KUKA KRL program: MyProgram_198().src

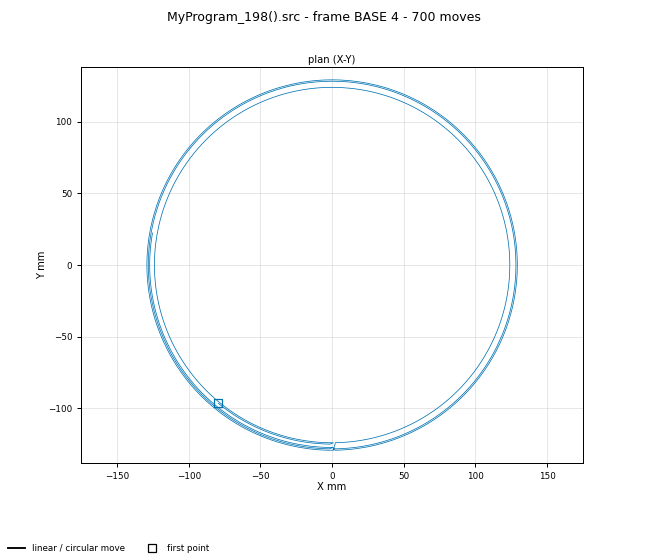
[picture p0: tool path of MyProgram_198().src in frame BASE 4, 700 of 700 moves have a stored position in this frame; points joined in program order, loops and branches not executed]
&ACCESS RVP
&REL 1
&PARAM TEMPLATE = C:\KRC\Roboter\Template\vorgabe
&PARAM EDITMASK = *
DEF MyProgram_198()
; ---- Setting reference (Base) ----
$BASE = BASE_DATA[4]

; --------------------------
; ---- Setting tool (TCP) ----
$TOOL = TOOL_DATA[3]
; --------------------------

$VEL.CP = VEL_APROX_PRINT
Startdeposition()
$VEL.CP = VEL_PRINT
LIN {X -79.3074,Y -96.5082,Z 142,A -131.7582,B 23.1277,C -1.1215,E1 23.053,E2 218.5929} C_DIS
LIN {X -76.0002,Y -99.1332,Z 142,A -129.8981,B 23.128,C -1.1147,E1 23.0571,E2 216.7428} C_DIS
LIN {X -73.2038,Y -101.2156,Z 142,A -128.0696,B 23.1276,C -1.1218,E1 23.0613,E2 214.889} C_DIS
LIN {X -68.9891,Y -104.1346,Z 142,A -125.8787,B 23.1281,C -1.111,E1 23.0663,E2 212.7178} C_DIS
LIN {X -65.7626,Y -106.2014,Z 142,A -124.3776,B 23.1288,C -1.0972,E1 23.0698,E2 211.2468} C_DIS
LIN {X -62.6284,Y -108.079,Z 142,A -122.461,B 23.1284,C -1.1052,E1 23.0744,E2 209.3034} C_DIS
LIN {X -59.0699,Y -110.0643,Z 142,A -120.3581,B 23.128,C -1.1129,E1 23.0796,E2 207.1744} C_DIS
LIN {X -55.3102,Y -111.9987,Z 142,A -118.661,B 23.1286,C -1.0998,E1 23.0838,E2 205.5056} C_DIS
LIN {X -52.0364,Y -113.5576,Z 142,A -116.9215,B 23.1286,C -1.1012,E1 23.0882,E2 203.7578} C_DIS
LIN {X -48.3423,Y -115.1781,Z 142,A -114.9515,B 23.1284,C -1.1045,E1 23.0933,E2 201.7745} C_DIS
LIN {X -44.2604,Y -116.8083,Z 142,A -113.1572,B 23.129,C -1.0928,E1 23.0979,E2 200.0059} C_DIS
LIN {X -41.267,Y -117.8988,Z 142,A -111.7171,B 23.129,C -1.0906,E1 23.1017,E2 198.5684} C_DIS
LIN {X -37.9757,Y -118.9992,Z 142,A -110.3261,B 23.1295,C -1.0804,E1 23.1053,E2 197.2004} C_DIS
LIN {X -34.3508,Y -120.098,Z 142,A -108.2397,B 23.1289,C -1.0946,E1 23.111,E2 195.0741} C_DIS
LIN {X -30.596,Y -121.1069,Z 142,A -106.5516,B 23.1291,C -1.0893,E1 23.1156,E2 193.3967} C_DIS
LIN {X -26.6613,Y -122.0338,Z 142,A -104.6727,B 23.1291,C -1.0895,E1 23.1207,E2 191.5148} C_DIS
LIN {X -23.1637,Y -122.7458,Z 142,A -102.9898,B 23.1291,C -1.0908,E1 23.1253,E2 189.8264} C_DIS
LIN {X -19.2282,Y -123.4232,Z 142,A -101.2648,B 23.1293,C -1.0855,E1 23.13,E2 188.1133} C_DIS
LIN {X -15.8715,Y -123.9001,Z 142,A -99.6847,B 23.1293,C -1.0863,E1 23.1344,E2 186.5299} C_DIS
LIN {X -11.9335,Y -124.3407,Z 142,A -97.8891,B 23.1293,C -1.0851,E1 23.1394,E2 184.7362} C_DIS
LIN {X -8.4853,Y -124.6251,Z 142,A -96.2436,B 23.1292,C -1.0876,E1 23.144,E2 183.0835} C_DIS
LIN {X -5.5832,Y -124.7887,Z 142,A -94.7991,B 23.129,C -1.0928,E1 23.1481,E2 181.6255} C_DIS
LIN {X -1.4686,Y -124.905,Z 142,A -92.9546,B 23.129,C -1.0911,E1 23.1532,E2 179.7852} C_DIS
LIN {X -1.4686,Y -124.905,Z 142,A -92.9546,B 23.129,C -1.0911,E1 23.1532,E2 179.7852} C_DIS
Enddeposition()
LIN {X 0.8717,Y -123.9392,Z 142,A -91.8325,B 22.3171,C -0.9594,E1 22.339,E2 178.8986} C_DIS
Startdeposition()
$VEL.CP = VEL_PRINT
LIN {X -2.2963,Y -123.9219,Z 142,A -93.916,B 22.3182,C -0.9325,E1 22.333,E2 181.0529} C_DIS
LIN {X -6.0852,Y -123.7935,Z 142,A -95.6272,B 22.3182,C -0.9341,E1 22.3282,E2 182.7603} C_DIS
LIN {X -9.1248,Y -123.6066,Z 142,A -97.0662,B 22.3182,C -0.9328,E1 22.3242,E2 184.2033} C_DIS
LIN {X -12.9239,Y -123.2677,Z 142,A -98.8033,B 22.3182,C -0.9341,E1 22.3194,E2 185.938} C_DIS
LIN {X -15.91,Y -122.9176,Z 142,A -100.1901,B 22.3182,C -0.9345,E1 22.3155,E2 187.3249} C_DIS
LIN {X -18.9628,Y -122.4836,Z 142,A -101.6065,B 22.3182,C -0.9352,E1 22.3116,E2 188.7406} C_DIS
LIN {X -21.9284,Y -121.9875,Z 142,A -103.0074,B 22.3182,C -0.9352,E1 22.3078,E2 190.1431} C_DIS
LIN {X -24.9422,Y -121.4073,Z 142,A -104.4213,B 22.3181,C -0.936,E1 22.3039,E2 191.5567} C_DIS
LIN {X -28.6367,Y -120.5898,Z 142,A -106.179,B 22.3181,C -0.9365,E1 22.2991,E2 193.3156} C_DIS
LIN {X -32.301,Y -119.6602,Z 142,A -107.9305,B 22.3181,C -0.9374,E1 22.2944,E2 195.0677} C_DIS
LIN {X -35.9945,Y -118.6012,Z 142,A -109.8524,B 22.3182,C -0.9326,E1 22.2892,E2 197.0059} C_DIS
LIN {X -40.3265,Y -117.199,Z 142,A -111.962,B 22.3182,C -0.9341,E1 22.2836,E2 199.116} C_DIS
LIN {X -43.9105,Y -115.9044,Z 142,A -113.5812,B 22.3178,C -0.9416,E1 22.2794,E2 200.7191} C_DIS
LIN {X -47.4374,Y -114.5057,Z 142,A -115.4966,B 22.318,C -0.9367,E1 22.2744,E2 202.6523} C_DIS
LIN {X -51.6487,Y -112.669,Z 142,A -117.6238,B 22.318,C -0.939,E1 22.269,E2 204.7794} C_DIS
LIN {X -55.3801,Y -110.8834,Z 142,A -119.4704,B 22.3178,C -0.944,E1 22.2644,E2 206.6182} C_DIS
LIN {X -58.4344,Y -109.3054,Z 142,A -120.9738,B 22.3175,C -0.9496,E1 22.2607,E2 208.1116} C_DIS
LIN {X -61.762,Y -107.4607,Z 142,A -122.9039,B 22.3177,C -0.945,E1 22.2559,E2 210.0601} C_DIS
LIN {X -65.6838,Y -105.1089,Z 142,A -125.0239,B 22.3176,C -0.9479,E1 22.2509,E2 212.1798} C_DIS
LIN {X -69.2138,Y -102.819,Z 142,A -126.9012,B 22.3174,C -0.9538,E1 22.2465,E2 214.0488} C_DIS
LIN {X -72.6168,Y -100.4441,Z 142,A -128.7387,B 22.3171,C -0.9603,E1 22.2424,E2 215.8762} C_DIS
LIN {X -75.6547,Y -98.1768,Z 142,A -130.6621,B 22.3172,C -0.9564,E1 22.238,E2 217.8175} C_DIS
LIN {X -79.2058,Y -95.3345,Z 142,A -132.6852,B 22.317,C -0.9636,E1 22.2337,E2 219.8305} C_DIS
LIN {X -82.3887,Y -92.5983,Z 142,A -134.734,B 22.317,C -0.963,E1 22.2293,E2 221.89} C_DIS
LIN {X -85.4698,Y -89.7616,Z 142,A -136.6617,B 22.3168,C -0.9673,E1 22.2254,E2 223.8153} C_DIS
LIN {X -88.7114,Y -86.5597,Z 142,A -138.7161,B 22.3165,C -0.9738,E1 22.2214,E2 225.8623} C_DIS
LIN {X -91.5742,Y -83.5252,Z 142,A -140.7246,B 22.3165,C -0.9749,E1 22.2176,E2 227.878} C_DIS
LIN {X -94.5817,Y -80.1033,Z 142,A -142.8001,B 22.3162,C -0.9809,E1 22.2138,E2 229.9482} C_DIS
LIN {X -96.7777,Y -77.4362,Z 142,A -144.4451,B 22.3162,C -0.9828,E1 22.2109,E2 231.597} C_DIS
LIN {X -99.5555,Y -73.8306,Z 142,A -146.5705,B 22.316,C -0.987,E1 22.2073,E2 233.7226} C_DIS
LIN {X -102.1996,Y -70.1244,Z 142,A -148.6828,B 22.3158,C -0.992,E1 22.2039,E2 235.8336} C_DIS
LIN {X -104.7148,Y -66.3102,Z 142,A -150.7774,B 22.3155,C -0.9981,E1 22.2007,E2 237.9239} C_DIS
LIN {X -106.7088,Y -63.0518,Z 142,A -152.5785,B 22.3154,C -1.0014,E1 22.1982,E2 239.7269} C_DIS
LIN {X -108.944,Y -59.1056,Z 142,A -154.6079,B 22.315,C -1.0097,E1 22.1954,E2 241.7464} C_DIS
LIN {X -110.5212,Y -56.0964,Z 142,A -156.1781,B 22.3148,C -1.0141,E1 22.1934,E2 243.3145} C_DIS
LIN {X -112.0468,Y -52.9856,Z 142,A -157.7322,B 22.3146,C -1.0204,E1 22.1915,E2 244.8615} C_DIS
LIN {X -113.6099,Y -49.5447,Z 142,A -159.6499,B 22.3146,C -1.0187,E1 22.1893,E2 246.7957} C_DIS
LIN {X -115.0085,Y -46.2039,Z 142,A -161.205,B 22.3142,C -1.0282,E1 22.1877,E2 248.3355} C_DIS
LIN {X -116.4356,Y -42.4819,Z 142,A -163.2031,B 22.3142,C -1.0275,E1 22.1857,E2 250.3482} C_DIS
LIN {X -117.9183,Y -38.1742,Z 142,A -165.3281,B 22.314,C -1.033,E1 22.1839,E2 252.4724} C_DIS
LIN {X -119.2482,Y -33.7908,Z 142,A -167.4478,B 22.3137,C -1.0393,E1 22.1822,E2 254.5893} C_DIS
LIN {X -120.2291,Y -30.1146,Z 142,A -169.1992,B 22.3135,C -1.045,E1 22.181,E2 256.3373} C_DIS
LIN {X -121.0983,Y -26.402,Z 142,A -170.8293,B 22.313,C -1.0555,E1 22.18,E2 257.9502} C_DIS
LIN {X -121.7047,Y -23.4477,Z 142,A -172.2411,B 22.3128,C -1.0592,E1 22.1792,E2 259.3619} C_DIS
LIN {X -122.2442,Y -20.449,Z 142,A -173.6444,B 22.3126,C -1.0637,E1 22.1785,E2 260.7624} C_DIS
LIN {X -122.7383,Y -17.2398,Z 142,A -175.2701,B 22.3126,C -1.0637,E1 22.1779,E2 262.3995} C_DIS
LIN {X -123.1888,Y -13.6572,Z 142,A -176.8563,B 22.3123,C -1.0721,E1 22.1774,E2 263.974} C_DIS
LIN {X -123.4861,Y -10.6336,Z 142,A -178.2667,B 22.3121,C -1.0763,E1 22.177,E2 265.3829} C_DIS
LIN {X -123.7095,Y -7.6032,Z 142,A -179.6751,B 22.3119,C -1.0806,E1 22.1767,E2 266.7895} C_DIS
LIN {X -123.8593,Y -4.5609,Z 142,A 178.7447,B 22.3119,C -1.0784,E1 22.1765,E2 268.3862} C_DIS
LIN {X -123.946,Y 0,Z 142,A 176.5529,B 22.3119,C -1.0819,E1 22.1765,E2 270.5837} C_DIS
LIN {X -123.8594,Y 4.5582,Z 142,A 174.6462,B 22.3111,C -1.0965,E1 22.1766,E2 272.4649} C_DIS
LIN {X -123.7172,Y 7.4784,Z 142,A 173.2388,B 22.3111,C -1.0986,E1 22.1768,E2 273.8762} C_DIS
LIN {X -123.4269,Y 11.3098,Z 142,A 171.3972,B 22.3109,C -1.1018,E1 22.1773,E2 275.7221} C_DIS
LIN {X -122.9987,Y 15.2809,Z 142,A 169.6572,B 22.3104,C -1.1118,E1 22.1778,E2 277.4473} C_DIS
LIN {X -122.5967,Y 18.2306,Z 142,A 168.2579,B 22.3102,C -1.1153,E1 22.1784,E2 278.8469} C_DIS
LIN {X -122.1586,Y 20.9622,Z 142,A 166.914,B 22.3102,C -1.1168,E1 22.179,E2 280.1957} C_DIS
LIN {X -121.5592,Y 24.1957,Z 142,A 165.4285,B 22.3099,C -1.123,E1 22.1798,E2 281.6749} C_DIS
LIN {X -120.93,Y 27.1649,Z 142,A 163.8565,B 22.3099,C -1.1209,E1 22.1807,E2 283.2629} C_DIS
LIN {X -119.8499,Y 31.5898,Z 142,A 161.7428,B 22.3097,C -1.1272,E1 22.1822,E2 285.3739} C_DIS
LIN {X -118.6079,Y 35.9727,Z 142,A 159.7772,B 22.3091,C -1.1392,E1 22.1837,E2 287.3206} C_DIS
LIN {X -117.6909,Y 38.8678,Z 142,A 158.2151,B 22.3091,C -1.1375,E1 22.185,E2 288.8976} C_DIS
LIN {X -116.4339,Y 42.4869,Z 142,A 156.5771,B 22.3087,C -1.148,E1 22.1866,E2 290.5181} C_DIS
LIN {X -115.0821,Y 46.0214,Z 142,A 154.664,B 22.3087,C -1.147,E1 22.1885,E2 292.446} C_DIS
LIN {X -113.3041,Y 50.2401,Z 142,A 152.519,B 22.3085,C -1.1523,E1 22.1909,E2 294.5905} C_DIS
LIN {X -111.72,Y 53.6698,Z 142,A 150.9241,B 22.3079,C -1.1633,E1 22.1928,E2 296.166} C_DIS
LIN {X -110.2395,Y 56.6497,Z 142,A 149.3135,B 22.3079,C -1.165,E1 22.1948,E2 297.7819} C_DIS
LIN {X -108.5935,Y 59.7474,Z 142,A 147.5881,B 22.3079,C -1.1657,E1 22.1971,E2 299.516} C_DIS
LIN {X -106.3109,Y 63.7204,Z 142,A 145.5115,B 22.3074,C -1.1733,E1 22.2,E2 301.5845} C_DIS
LIN {X -104.2933,Y 66.9711,Z 142,A 143.6733,B 22.3074,C -1.1755,E1 22.2028,E2 303.4275} C_DIS
LIN {X -101.7782,Y 70.7347,Z 142,A 141.5651,B 22.3071,C -1.1807,E1 22.2061,E2 305.5339} C_DIS
LIN {X -99.0918,Y 74.4518,Z 142,A 139.6016,B 22.3065,C -1.1925,E1 22.2093,E2 307.477} C_DIS
LIN {X -96.7618,Y 77.4562,Z 142,A 137.6837,B 22.3065,C -1.1908,E1 22.2126,E2 309.4096} C_DIS
LIN {X -94.1026,Y 80.6658,Z 142,A 135.7295,B 22.3063,C -1.1946,E1 22.2162,E2 311.3637} C_DIS
LIN {X -91.0649,Y 84.08,Z 142,A 133.6742,B 22.306,C -1.2021,E1 22.22,E2 313.4095} C_DIS
LIN {X -88.1717,Y 87.1095,Z 142,A 131.6512,B 22.306,C -1.2034,E1 22.2239,E2 315.4391} C_DIS
LIN {X -85.1819,Y 90.0348,Z 142,A 129.7181,B 22.3057,C -1.208,E1 22.2278,E2 317.3691} C_DIS
LIN {X -81.817,Y 93.1037,Z 142,A 127.6556,B 22.3053,C -1.2144,E1 22.2321,E2 319.424} C_DIS
LIN {X -78.9119,Y 95.5779,Z 142,A 125.9078,B 22.3051,C -1.2189,E1 22.2358,E2 321.1675} C_DIS
LIN {X -75.653,Y 98.1781,Z 142,A 123.875,B 22.3051,C -1.2188,E1 22.2403,E2 323.2091} C_DIS
LIN {X -71.9821,Y 100.8999,Z 142,A 121.7591,B 22.3049,C -1.2229,E1 22.2451,E2 325.3224} C_DIS
LIN {X -68.2096,Y 103.4874,Z 142,A 119.7612,B 22.3044,C -1.2317,E1 22.2497,E2 327.3049} C_DIS
LIN {X -64.9188,Y 105.583,Z 142,A 117.827,B 22.3045,C -1.2298,E1 22.2543,E2 329.2509} C_DIS
LIN {X -61.0554,Y 107.8637,Z 142,A 115.7414,B 22.3044,C -1.2329,E1 22.2593,E2 331.3353} C_DIS
LIN {X -57.2646,Y 109.9211,Z 142,A 113.8732,B 22.3039,C -1.2413,E1 22.2639,E2 333.1873} C_DIS
LIN {X -54.3534,Y 111.3899,Z 142,A 112.3781,B 22.3038,C -1.2441,E1 22.2676,E2 334.6793} C_DIS
LIN {X -51.6084,Y 112.6876,Z 142,A 110.971,B 22.3037,C -1.2461,E1 22.2712,E2 336.0852} C_DIS
LIN {X -48.1162,Y 114.2222,Z 142,A 109.0475,B 22.3039,C -1.2422,E1 22.2761,E2 338.0243} C_DIS
LIN {X -44.599,Y 115.6408,Z 142,A 107.3018,B 22.3037,C -1.2448,E1 22.2807,E2 339.7673} C_DIS
LIN {X -40.9841,Y 116.971,Z 142,A 105.5035,B 22.3037,C -1.2463,E1 22.2854,E2 341.5657} C_DIS
LIN {X -36.678,Y 118.392,Z 142,A 103.3984,B 22.3036,C -1.2483,E1 22.291,E2 343.6697} C_DIS
LIN {X -33.0611,Y 119.4523,Z 142,A 101.6561,B 22.3035,C -1.2501,E1 22.2957,E2 345.4105} C_DIS
LIN {X -28.6324,Y 120.5908,Z 142,A 99.5287,B 22.3034,C -1.2515,E1 22.3014,E2 347.5374} C_DIS
LIN {X -24.94,Y 121.4078,Z 142,A 97.9393,B 22.303,C -1.2595,E1 22.3057,E2 349.108} C_DIS
LIN {X -21.8511,Y 122.0014,Z 142,A 96.4534,B 22.303,C -1.2593,E1 22.3098,E2 350.5964} C_DIS
LIN {X -18.1786,Y 122.6042,Z 142,A 94.7493,B 22.3029,C -1.2611,E1 22.3145,E2 352.2975} C_DIS
LIN {X -15.1689,Y 123.0121,Z 142,A 93.1894,B 22.3032,C -1.2555,E1 22.3189,E2 353.8733} C_DIS
LIN {X -11.0173,Y 123.4536,Z 142,A 91.3043,B 22.303,C -1.2582,E1 22.3241,E2 355.7524} C_DIS
LIN {X -7.5913,Y 123.7102,Z 142,A 89.8371,B 22.3027,C -1.2639,E1 22.3281,E2 357.2053} C_DIS
LIN {X -4.5569,Y 123.8595,Z 142,A 88.2717,B 22.3031,C -1.2576,E1 22.3325,E2 358.7875} C_DIS
LIN {X -0.7453,Y 123.9408,Z 142,A 86.6712,B 22.3027,C -1.2647,E1 22.337,E2 360.3694} C_DIS
LIN {X 2.3024,Y 123.9218,Z 142,A 85.1012,B 22.303,C -1.2582,E1 22.3414,E2 361.9564} C_DIS
LIN {X 6.8655,Y 123.7543,Z 142,A 83.1554,B 22.3027,C -1.2651,E1 22.3468,E2 363.8832} C_DIS
LIN {X 9.895,Y 123.5484,Z 142,A 81.7369,B 22.3027,C -1.2644,E1 22.3507,E2 365.3028} C_DIS
LIN {X 12.9191,Y 123.2682,Z 142,A 80.2409,B 22.3029,C -1.2603,E1 22.3549,E2 366.8084} C_DIS
LIN {X 16.5992,Y 122.8272,Z 142,A 78.473,B 22.3031,C -1.2576,E1 22.3598,E2 368.5818} C_DIS
LIN {X 20.4296,Y 122.2475,Z 142,A 76.8358,B 22.3027,C -1.2635,E1 22.3643,E2 370.2016} C_DIS
LIN {X 23.5219,Y 121.6905,Z 142,A 75.2611,B 22.3031,C -1.2578,E1 22.3686,E2 371.7896} C_DIS
LIN {X 27.4214,Y 120.8714,Z 142,A 73.4485,B 22.3031,C -1.2581,E1 22.3736,E2 373.5987} C_DIS
LIN {X 31.608,Y 119.845,Z 142,A 71.4007,B 22.3032,C -1.2545,E1 22.3791,E2 375.6523} C_DIS
LIN {X 35.9885,Y 118.603,Z 142,A 69.3051,B 22.3032,C -1.2533,E1 22.3848,E2 377.7469} C_DIS
LIN {X 40.3212,Y 117.2009,Z 142,A 67.3524,B 22.303,C -1.2581,E1 22.3899,E2 379.6829} C_DIS
LIN {X 43.3345,Y 116.1202,Z 142,A 65.7635,B 22.3034,C -1.252,E1 22.3941,E2 381.2839} C_DIS
LIN {X 46.7481,Y 114.7892,Z 142,A 64.0309,B 22.3035,C -1.2486,E1 22.3986,E2 383.021} C_DIS
LIN {X 50.936,Y 112.9928,Z 142,A 62.0812,B 22.3033,C -1.253,E1 22.4035,E2 384.9539} C_DIS
LIN {X 53.6652,Y 111.7222,Z 142,A 60.6564,B 22.3035,C -1.2499,E1 22.4071,E2 386.3827} C_DIS
LIN {X 57.0846,Y 110.0156,Z 142,A 58.9614,B 22.3035,C -1.2507,E1 22.4113,E2 388.0703} C_DIS
LIN {X 60.4301,Y 108.2151,Z 142,A 57.0274,B 22.304,C -1.2405,E1 22.4161,E2 390.0246} C_DIS
LIN {X 64.3888,Y 105.9073,Z 142,A 54.9005,B 22.3042,C -1.237,E1 22.4212,E2 392.1533} C_DIS
LIN {X 68.2553,Y 103.4573,Z 142,A 52.8091,B 22.3042,C -1.2347,E1 22.4261,E2 394.243} C_DIS
LIN {X 71.9872,Y 100.8962,Z 142,A 50.7274,B 22.3044,C -1.2316,E1 22.4309,E2 396.3246} C_DIS
LIN {X 75.6425,Y 98.1863,Z 142,A 48.6243,B 22.3046,C -1.2279,E1 22.4356,E2 398.4288} C_DIS
LIN {X 79.2139,Y 95.3278,Z 142,A 46.6078,B 22.3046,C -1.2282,E1 22.4399,E2 400.4358} C_DIS
LIN {X 82.4003,Y 92.588,Z 142,A 44.5842,B 22.305,C -1.2208,E1 22.4442,E2 402.4698} C_DIS
LIN {X 85.4671,Y 89.7642,Z 142,A 42.6802,B 22.3052,C -1.2179,E1 22.4481,E2 404.3726} C_DIS
LIN {X 88.7091,Y 86.5621,Z 142,A 40.6465,B 22.3052,C -1.2166,E1 22.4521,E2 406.3999} C_DIS
LIN {X 91.5695,Y 83.5304,Z 142,A 38.6578,B 22.3056,C -1.2095,E1 22.4559,E2 408.3972} C_DIS
LIN {X 94.591,Y 80.0924,Z 142,A 36.6269,B 22.3056,C -1.2084,E1 22.4596,E2 410.4206} C_DIS
LIN {X 97.2514,Y 76.8407,Z 142,A 34.6896,B 22.3059,C -1.204,E1 22.463,E2 412.3592} C_DIS
LIN {X 99.5507,Y 73.837,Z 142,A 32.8768,B 22.3062,C -1.1969,E1 22.466,E2 414.1809} C_DIS
LIN {X 102.2052,Y 70.1163,Z 142,A 30.783,B 22.3065,C -1.1924,E1 22.4694,E2 416.2748} C_DIS
LIN {X 104.4189,Y 66.775,Z 142,A 28.9924,B 22.3065,C -1.1904,E1 22.4721,E2 418.0605} C_DIS
LIN {X 106.719,Y 63.0344,Z 142,A 26.9374,B 22.3069,C -1.1839,E1 22.4751,E2 420.1206} C_DIS
LIN {X 108.9413,Y 59.1106,Z 142,A 24.9414,B 22.3069,C -1.1823,E1 22.4778,E2 422.1091} C_DIS
LIN {X 110.3519,Y 56.4289,Z 142,A 23.6107,B 22.307,C -1.1816,E1 22.4795,E2 423.4336} C_DIS
LIN {X 111.7602,Y 53.5856,Z 142,A 22.0436,B 22.3074,C -1.173,E1 22.4814,E2 425.0138} C_DIS
LIN {X 113.3091,Y 50.2289,Z 142,A 20.4626,B 22.3074,C -1.1739,E1 22.4832,E2 426.5826} C_DIS
LIN {X 114.7964,Y 46.73,Z 142,A 18.555,B 22.308,C -1.162,E1 22.4853,E2 428.5093} C_DIS
LIN {X 116.4347,Y 42.4845,Z 142,A 16.4589,B 22.3083,C -1.1562,E1 22.4873,E2 430.6074} C_DIS
LIN {X 117.9158,Y 38.1821,Z 142,A 14.5324,B 22.3082,C -1.1579,E1 22.489,E2 432.517} C_DIS
LIN {X 118.9989,Y 34.6564,Z 142,A 12.8155,B 22.3085,C -1.1523,E1 22.4904,E2 434.2377} C_DIS
LIN {X 120.0323,Y 30.8902,Z 142,A 10.8916,B 22.309,C -1.1414,E1 22.4918,E2 436.1774} C_DIS
LIN {X 121.0928,Y 26.4273,Z 142,A 8.9201,B 22.309,C -1.1416,E1 22.493,E2 438.1353} C_DIS
LIN {X 121.8497,Y 22.6894,Z 142,A 7.0741,B 22.3094,C -1.1324,E1 22.494,E2 439.9934} C_DIS
LIN {X 122.4848,Y 18.955,Z 142,A 5.425,B 22.3094,C -1.1315,E1 22.4948,E2 441.6337} C_DIS
LIN {X 123.0119,Y 15.1704,Z 142,A 3.6994,B 22.3097,C -1.1278,E1 22.4954,E2 443.3574} C_DIS
LIN {X 123.3462,Y 12.1505,Z 142,A 2.3087,B 22.3098,C -1.124,E1 22.4958,E2 444.7488} C_DIS
LIN {X 123.621,Y 8.9269,Z 142,A 0.7565,B 22.3102,C -1.1167,E1 22.4961,E2 446.3096} C_DIS
LIN {X 123.8594,Y 4.5572,Z 142,A -1.3319,B 22.3106,C -1.1073,E1 22.4964,E2 448.4087} C_DIS
LIN {X 123.9459,Y 0.017,Z 142,A -3.3195,B 22.3107,C -1.1056,E1 22.4964,E2 450.3872} C_DIS
LIN {X 123.9065,Y -3.0353,Z 142,A -4.6782,B 22.3108,C -1.1035,E1 22.4964,E2 451.7422} C_DIS
LIN {X 123.7935,Y -6.0869,Z 142,A -6.0652,B 22.311,C -1.1001,E1 22.4962,E2 453.1288} C_DIS
LIN {X 123.5826,Y -9.4536,Z 142,A -7.6911,B 22.3113,C -1.092,E1 22.4959,E2 454.7649} C_DIS
LIN {X 123.2685,Y -12.9166,Z 142,A -9.2129,B 22.3113,C -1.0908,E1 22.4955,E2 456.2796} C_DIS
LIN {X 122.8178,Y -16.671,Z 142,A -10.9283,B 22.3116,C -1.0867,E1 22.4949,E2 457.9943} C_DIS
LIN {X 122.3704,Y -19.6926,Z 142,A -12.3232,B 22.3118,C -1.083,E1 22.4943,E2 459.3897} C_DIS
LIN {X 121.812,Y -22.8863,Z 142,A -13.9781,B 22.3123,C -1.0711,E1 22.4935,E2 461.0647} C_DIS
LIN {X 120.9197,Y -27.21,Z 142,A -16.008,B 22.3126,C -1.0651,E1 22.4923,E2 463.0968} C_DIS
LIN {X 119.8492,Y -31.5924,Z 142,A -18.0816,B 22.3128,C -1.0591,E1 22.4909,E2 465.1727} C_DIS
LIN {X 118.604,Y -35.9854,Z 142,A -20.0205,B 22.3128,C -1.0603,E1 22.4894,E2 467.0958} C_DIS
LIN {X 117.6877,Y -38.8773,Z 142,A -21.4155,B 22.313,C -1.0563,E1 22.4882,E2 468.4922} C_DIS
LIN {X 116.6962,Y -41.7592,Z 142,A -22.9368,B 22.3134,C -1.0468,E1 22.4867,E2 470.0288} C_DIS
LIN {X 115.3575,Y -45.3276,Z 142,A -24.7206,B 22.3137,C -1.0404,E1 22.4849,E2 471.8181} C_DIS
LIN {X 113.6147,Y -49.5335,Z 142,A -26.7981,B 22.3139,C -1.0353,E1 22.4827,E2 473.8961} C_DIS
LIN {X 111.9515,Y -53.1852,Z 142,A -28.6043,B 22.3141,C -1.032,E1 22.4805,E2 475.6999} C_DIS
LIN {X 110.3004,Y -56.5301,Z 142,A -30.2933,B 22.3142,C -1.0285,E1 22.4784,E2 477.3878} C_DIS
LIN {X 108.581,Y -59.77,Z 142,A -32.0443,B 22.3145,C -1.021,E1 22.4761,E2 479.1479} C_DIS
LIN {X 106.3109,Y -63.7204,Z 142,A -34.1443,B 22.3148,C -1.0152,E1 22.4731,E2 481.2507} C_DIS
LIN {X 103.8834,Y -67.6051,Z 142,A -36.2396,B 22.315,C -1.0103,E1 22.47,E2 483.347} C_DIS
LIN {X 101.3314,Y -71.3733,Z 142,A -38.3243,B 22.3152,C -1.0054,E1 22.4667,E2 485.4329} C_DIS
LIN {X 98.6425,Y -75.0463,Z 142,A -40.4278,B 22.3154,C -0.9998,E1 22.4631,E2 487.5397} C_DIS
LIN {X 95.7941,Y -78.6496,Z 142,A -42.4577,B 22.3155,C -0.9984,E1 22.4596,E2 489.5625} C_DIS
LIN {X 93.1031,Y -81.8177,Z 142,A -44.3785,B 22.3157,C -0.9935,E1 22.4561,E2 491.4862} C_DIS
LIN {X 90.5128,Y -84.6741,Z 142,A -46.1372,B 22.3159,C -0.9902,E1 22.4528,E2 493.245} C_DIS
LIN {X 87.6214,Y -87.6631,Z 142,A -48.129,B 22.3162,C -0.9824,E1 22.4488,E2 495.2475} C_DIS
LIN {X 84.6231,Y -90.5603,Z 142,A -50.0304,B 22.3163,C -0.979,E1 22.445,E2 497.1488} C_DIS
LIN {X 81.216,Y -93.6284,Z 142,A -52.157,B 22.3165,C -0.9738,E1 22.4405,E2 499.2794} C_DIS
LIN {X 78.0288,Y -96.3004,Z 142,A -54.0561,B 22.3167,C -0.9707,E1 22.4364,E2 501.1785} C_DIS
LIN {X 74.453,Y -99.0909,Z 142,A -56.1566,B 22.3169,C -0.9661,E1 22.4318,E2 503.2824} C_DIS
LIN {X 70.743,Y -101.7724,Z 142,A -58.2583,B 22.317,C -0.9624,E1 22.427,E2 505.3854} C_DIS
LIN {X 66.9581,Y -104.3016,Z 142,A -60.3509,B 22.3171,C -0.9589,E1 22.4221,E2 507.4794} C_DIS
LIN {X 63.0567,Y -106.7059,Z 142,A -62.4551,B 22.3173,C -0.9557,E1 22.4171,E2 509.5846} C_DIS
LIN {X 59.118,Y -108.9373,Z 142,A -64.5655,B 22.3175,C -0.9512,E1 22.4119,E2 511.6996} C_DIS
LIN {X 55.2848,Y -110.9304,Z 142,A -66.4642,B 22.3175,C -0.9523,E1 22.4072,E2 513.5895} C_DIS
LIN {X 51.6616,Y -112.663,Z 142,A -68.2372,B 22.3174,C -0.9532,E1 22.4027,E2 515.3552} C_DIS
LIN {X 48.1088,Y -114.2253,Z 142,A -70.1701,B 22.3177,C -0.9444,E1 22.3977,E2 517.3058} C_DIS
LIN {X 43.9118,Y -115.9039,Z 142,A -72.1075,B 22.3176,C -0.9483,E1 22.3927,E2 519.2283} C_DIS
LIN {X 40.3106,Y -117.2045,Z 142,A -74.0028,B 22.3179,C -0.9405,E1 22.3877,E2 521.1394} C_DIS
LIN {X 36.7007,Y -118.3851,Z 142,A -75.7769,B 22.318,C -0.9377,E1 22.383,E2 522.9173} C_DIS
LIN {X 33.0811,Y -119.4467,Z 142,A -77.354,B 22.3178,C -0.9431,E1 22.3788,E2 524.4773} C_DIS
LIN {X 29.3499,Y -120.4179,Z 142,A -79.1334,B 22.3178,C -0.9414,E1 22.374,E2 526.2579} C_DIS
LIN {X 25.665,Y -121.2574,Z 142,A -80.8674,B 22.3178,C -0.9404,E1 22.3692,E2 527.992} C_DIS
LIN {X 22.6853,Y -121.8505,Z 142,A -82.2664,B 22.3179,C -0.9395,E1 22.3654,E2 529.3915} C_DIS
LIN {X 19.214,Y -122.4447,Z 142,A -83.9711,B 22.3181,C -0.935,E1 22.3607,E2 531.1061} C_DIS
LIN {X 15.3695,Y -122.9881,Z 142,A -85.7751,B 22.3181,C -0.9335,E1 22.3557,E2 532.9124} C_DIS
LIN {X 12.1455,Y -123.3467,Z 142,A -87.1981,B 22.3181,C -0.936,E1 22.3518,E2 534.3277} C_DIS
LIN {X 8.8298,Y -123.6281,Z 142,A -88.793,B 22.3181,C -0.9328,E1 22.3473,E2 535.93} C_DIS
LIN {X 5.287,Y -123.831,Z 142,A -90.3796,B 22.3181,C -0.9345,E1 22.3429,E2 537.5115} C_DIS
LIN {X 2.2861,Y -123.9221,Z 142,A -91.7661,B 22.3181,C -0.9342,E1 22.339,E2 538.8986} C_DIS
LIN {X 2.2861,Y -123.9221,Z 142,A -91.7661,B 22.3181,C -0.9342,E1 22.339,E2 538.8986} C_DIS
Enddeposition()
LIN {X 0.9159,Y -129.1721,Z 143,A -92.6978,B 24.9656,C -1.3555,E1 25.0017,E2 539.1265} C_DIS
Startdeposition()
$VEL.CP = VEL_PRINT
LIN {X -2.056,Y -129.1619,Z 143,A -94.4314,B 24.9667,C -1.3341,E1 24.9968,E2 540.9106} C_DIS
LIN {X -5.4479,Y -129.064,Z 143,A -95.9238,B 24.9667,C -1.3346,E1 24.9926,E2 542.4023} C_DIS
LIN {X -9.2404,Y -128.8474,Z 143,A -97.6422,B 24.9667,C -1.3329,E1 24.9878,E2 544.1253} C_DIS
LIN {X -12.7283,Y -128.5501,Z 143,A -99.1732,B 24.9667,C -1.334,E1 24.9835,E2 545.6542} C_DIS
LIN {X -16.3368,Y -128.1417,Z 143,A -100.8519,B 24.9668,C -1.3309,E1 24.9789,E2 547.3415} C_DIS
LIN {X -19.8619,Y -127.642,Z 143,A -102.343,B 24.9666,C -1.3357,E1 24.9748,E2 548.8224} C_DIS
LIN {X -22.8537,Y -127.1404,Z 143,A -103.6917,B 24.9666,C -1.336,E1 24.9711,E2 550.1718} C_DIS
LIN {X -25.8549,Y -126.5642,Z 143,A -105.0506,B 24.9666,C -1.3364,E1 24.9673,E2 551.5314} C_DIS
LIN {X -28.9111,Y -125.9012,Z 143,A -106.4793,B 24.9666,C -1.335,E1 24.9634,E2 552.9651} C_DIS
LIN {X -32.1688,Y -125.109,Z 143,A -107.9331,B 24.9665,C -1.3375,E1 24.9595,E2 554.4151} C_DIS
LIN {X -35.1544,Y -124.303,Z 143,A -109.3333,B 24.9665,C -1.337,E1 24.9557,E2 555.8187} C_DIS
LIN {X -38.1245,Y -123.4243,Z 143,A -110.714,B 24.9665,C -1.3377,E1 24.952,E2 557.2001} C_DIS
LIN {X -41.0909,Y -122.4685,Z 143,A -112.1194,B 24.9665,C -1.3377,E1 24.9483,E2 558.6082} C_DIS
LIN {X -44.1762,Y -121.3899,Z 143,A -113.5097,B 24.9663,C -1.3418,E1 24.9447,E2 559.9913} C_DIS
LIN {X -47.0009,Y -120.324,Z 143,A -114.8983,B 24.9663,C -1.3407,E1 24.941,E2 561.3855} C_DIS
LIN {X -50.1973,Y -119.0266,Z 143,A -116.3763,B 24.9661,C -1.3449,E1 24.9372,E2 562.857} C_DIS
LIN {X -52.9783,Y -117.8145,Z 143,A -117.7771,B 24.9661,C -1.3437,E1 24.9336,E2 564.2639} C_DIS
LIN {X -55.9912,Y -116.413,Z 143,A -119.242,B 24.9661,C -1.3459,E1 24.9299,E2 565.7273} C_DIS
LIN {X -59.3318,Y -114.7488,Z 143,A -120.895,B 24.966,C -1.3481,E1 24.9258,E2 567.3795} C_DIS
LIN {X -62.0674,Y -113.2919,Z 143,A -122.3372,B 24.966,C -1.3467,E1 24.9223,E2 568.8291} C_DIS
LIN {X -65.7504,Y -111.1953,Z 143,A -124.2414,B 24.966,C -1.3482,E1 24.9177,E2 570.7353} C_DIS
LIN {X -69.2992,Y -109.0191,Z 143,A -126.1244,B 24.9659,C -1.3493,E1 24.9132,E2 572.6217} C_DIS
LIN {X -72.7546,Y -106.7441,Z 143,A -127.9389,B 24.9657,C -1.3533,E1 24.909,E2 574.4326} C_DIS
LIN {X -76.1455,Y -104.3523,Z 143,A -129.8434,B 24.9657,C -1.3534,E1 24.9047,E2 576.3436} C_DIS
LIN {X -79.5443,Y -101.7849,Z 143,A -131.7274,B 24.9655,C -1.3571,E1 24.9005,E2 578.2255} C_DIS
LIN {X -82.9887,Y -98.9962,Z 143,A -133.656,B 24.9652,C -1.3627,E1 24.8963,E2 580.1483} C_DIS
LIN {X -86.0043,Y -96.3882,Z 143,A -135.4758,B 24.9652,C -1.3638,E1 24.8925,E2 581.9727} C_DIS
LIN {X -89.2124,Y -93.4265,Z 143,A -137.3778,B 24.9649,C -1.3695,E1 24.8887,E2 583.8689} C_DIS
LIN {X -92.1442,Y -90.5364,Z 143,A -139.2175,B 24.9647,C -1.3728,E1 24.885,E2 585.7086} C_DIS
LIN {X -95.0674,Y -87.4617,Z 143,A -141.1028,B 24.9645,C -1.3768,E1 24.8814,E2 587.5924} C_DIS
LIN {X -97.7978,Y -84.3977,Z 143,A -142.9421,B 24.9643,C -1.3802,E1 24.878,E2 589.4321} C_DIS
LIN {X -100.3934,Y -81.2933,Z 143,A -144.781,B 24.9643,C -1.3824,E1 24.8748,E2 591.2742} C_DIS
LIN {X -103.1453,Y -77.7716,Z 143,A -146.7048,B 24.9638,C -1.3901,E1 24.8715,E2 593.189} C_DIS
LIN {X -105.593,Y -74.4143,Z 143,A -148.5941,B 24.9637,C -1.3926,E1 24.8684,E2 595.0815} C_DIS
LIN {X -108.1233,Y -70.6887,Z 143,A -150.6532,B 24.9636,C -1.3949,E1 24.8652,E2 597.1453} C_DIS
LIN {X -110.5126,Y -66.8905,Z 143,A -152.5862,B 24.9631,C -1.4029,E1 24.8624,E2 599.0691} C_DIS
LIN {X -112.6373,Y -63.2473,Z 143,A -154.4442,B 24.9628,C -1.4087,E1 24.8598,E2 600.9231} C_DIS
LIN {X -114.6313,Y -59.5554,Z 143,A -156.2326,B 24.9624,C -1.4173,E1 24.8575,E2 602.7004} C_DIS
LIN {X -115.9907,Y -56.8607,Z 143,A -157.6515,B 24.9624,C -1.4173,E1 24.8557,E2 604.1268} C_DIS
LIN {X -117.3701,Y -53.9558,Z 143,A -159.0627,B 24.9621,C -1.4222,E1 24.8541,E2 605.5342} C_DIS
LIN {X -118.7433,Y -50.8635,Z 143,A -160.5441,B 24.9618,C -1.4275,E1 24.8524,E2 607.0112} C_DIS
LIN {X -119.9639,Y -47.9137,Z 143,A -161.9681,B 24.9616,C -1.4313,E1 24.8509,E2 608.434} C_DIS
LIN {X -121.2134,Y -44.6621,Z 143,A -163.5143,B 24.9614,C -1.4359,E1 24.8494,E2 609.978} C_DIS
LIN {X -122.134,Y -42.0745,Z 143,A -164.8037,B 24.9614,C -1.4363,E1 24.8482,E2 611.2738} C_DIS
LIN {X -123.292,Y -38.5568,Z 143,A -166.4004,B 24.961,C -1.4434,E1 24.8468,E2 612.8627} C_DIS
LIN {X -124.1938,Y -35.545,Z 143,A -167.8019,B 24.9608,C -1.4474,E1 24.8457,E2 614.2628} C_DIS
LIN {X -125.2569,Y -31.5861,Z 143,A -169.6431,B 24.9605,C -1.452,E1 24.8444,E2 616.1037} C_DIS
LIN {X -125.956,Y -28.6712,Z 143,A -170.9863,B 24.9603,C -1.4556,E1 24.8436,E2 617.4462} C_DIS
LIN {X -126.7368,Y -25.0066,Z 143,A -172.6367,B 24.96,C -1.4614,E1 24.8427,E2 619.0926} C_DIS
LIN {X -127.1856,Y -22.6012,Z 143,A -173.7503,B 24.9599,C -1.4636,E1 24.8421,E2 620.2076} C_DIS
LIN {X -127.7607,Y -19.0953,Z 143,A -175.3051,B 24.9595,C -1.4696,E1 24.8414,E2 621.7572} C_DIS
LIN {X -128.2196,Y -15.7127,Z 143,A -176.9142,B 24.9595,C -1.4701,E1 24.8408,E2 623.3748} C_DIS
LIN {X -128.5897,Y -12.3156,Z 143,A -178.3686,B 24.9591,C -1.4779,E1 24.8404,E2 624.8194} C_DIS
LIN {X -128.8707,Y -8.9214,Z 143,A 179.9612,B 24.9592,C -1.4754,E1 24.8401,E2 626.5054} C_DIS
LIN {X -129.0837,Y -4.9409,Z 143,A 178.2793,B 24.9587,C -1.4852,E1 24.8399,E2 628.1742} C_DIS
LIN {X -129.1779,Y -0.7281,Z 143,A 176.5535,B 24.958,C -1.4979,E1 24.8398,E2 629.88} C_DIS
LIN {X -129.1484,Y 2.8673,Z 143,A 174.6921,B 24.9584,C -1.4909,E1 24.8398,E2 631.7694} C_DIS
LIN {X -129.0162,Y 6.4677,Z 143,A 173.2186,B 24.9577,C -1.5019,E1 24.84,E2 633.2255} C_DIS
LIN {X -128.8182,Y 9.6396,Z 143,A 171.6973,B 24.9577,C -1.5014,E1 24.8403,E2 634.7572} C_DIS
LIN {X -128.447,Y 13.7243,Z 143,A 169.9891,B 24.9571,C -1.5125,E1 24.8408,E2 636.4492} C_DIS
LIN {X -128.0706,Y 16.8793,Z 143,A 168.6059,B 24.9568,C -1.5183,E1 24.8413,E2 637.8267} C_DIS
LIN {X -127.642,Y 19.8619,Z 143,A 167.2193,B 24.9567,C -1.5204,E1 24.8418,E2 639.2165} C_DIS
LIN {X -127.1488,Y 22.8066,Z 143,A 165.8698,B 24.9565,C -1.5236,E1 24.8425,E2 640.5665} C_DIS
LIN {X -126.4956,Y 26.1918,Z 143,A 164.3438,B 24.9562,C -1.5287,E1 24.8433,E2 642.0893} C_DIS
LIN {X -125.7625,Y 29.5184,Z 143,A 162.8181,B 24.956,C -1.5329,E1 24.8443,E2 643.6139} C_DIS
LIN {X -125.124,Y 32.1099,Z 143,A 161.6132,B 24.9558,C -1.5358,E1 24.8451,E2 644.819} C_DIS
LIN {X -124.2571,Y 35.3187,Z 143,A 160.13,B 24.9556,C -1.5402,E1 24.8462,E2 646.3005} C_DIS
LIN {X -123.292,Y 38.5568,Z 143,A 158.6267,B 24.9553,C -1.5447,E1 24.8474,E2 647.8016} C_DIS
LIN {X -122.392,Y 41.3207,Z 143,A 157.3124,B 24.9551,C -1.5477,E1 24.8486,E2 649.1162} C_DIS
LIN {X -121.2507,Y 44.5625,Z 143,A 155.7902,B 24.9548,C -1.5526,E1 24.85,E2 650.6354} C_DIS
LIN {X -120.3028,Y 47.0554,Z 143,A 154.5682,B 24.9548,C -1.5546,E1 24.8512,E2 651.8597} C_DIS
LIN {X -119.1061,Y 50.0069,Z 143,A 153.1534,B 24.9545,C -1.5589,E1 24.8527,E2 653.2721} C_DIS
LIN {X -117.8285,Y 52.9469,Z 143,A 151.726,B 24.9542,C -1.563,E1 24.8543,E2 654.6975} C_DIS
LIN {X -116.2564,Y 56.3189,Z 143,A 150.0863,B 24.9539,C -1.5685,E1 24.8563,E2 656.333} C_DIS
LIN {X -114.8669,Y 59.0997,Z 143,A 148.6757,B 24.9537,C -1.5712,E1 24.8581,E2 657.7447} C_DIS
LIN {X -113.0365,Y 62.5309,Z 143,A 146.8533,B 24.9537,C -1.5718,E1 24.8605,E2 659.5752} C_DIS
LIN {X -110.7887,Y 66.4331,Z 143,A 144.8237,B 24.9534,C -1.5762,E1 24.8634,E2 661.6048} C_DIS
LIN {X -108.5736,Y 69.9951,Z 143,A 142.9857,B 24.9531,C -1.5826,E1 24.8661,E2 663.4369} C_DIS
LIN {X -106.275,Y 73.4381,Z 143,A 141.0995,B 24.9529,C -1.5855,E1 24.8691,E2 665.3256} C_DIS
LIN {X -103.7633,Y 76.9455,Z 143,A 139.1694,B 24.9526,C -1.5901,E1 24.8723,E2 667.2542} C_DIS
LIN {X -101.1059,Y 80.405,Z 143,A 137.2778,B 24.9522,C -1.5973,E1 24.8755,E2 669.1375} C_DIS
LIN {X -98.3881,Y 83.7087,Z 143,A 135.3825,B 24.9519,C -1.6025,E1 24.8789,E2 671.0293} C_DIS
LIN {X -95.7067,Y 86.7618,Z 143,A 133.5496,B 24.9517,C -1.6057,E1 24.8823,E2 672.8626} C_DIS
LIN {X -92.8819,Y 89.7794,Z 143,A 131.693,B 24.9515,C -1.6092,E1 24.8859,E2 674.7189} C_DIS
LIN {X -89.8928,Y 92.7721,Z 143,A 129.8186,B 24.9512,C -1.6139,E1 24.8896,E2 676.5901} C_DIS
LIN {X -86.8984,Y 95.5827,Z 143,A 127.9763,B 24.951,C -1.6173,E1 24.8934,E2 678.4319} C_DIS
LIN {X -83.7087,Y 98.3881,Z 143,A 126.0947,B 24.9507,C -1.6217,E1 24.8973,E2 680.3102} C_DIS
LIN {X -80.405,Y 101.1059,Z 143,A 124.2112,B 24.9504,C -1.6266,E1 24.9014,E2 682.1892} C_DIS
LIN {X -77.1058,Y 103.6439,Z 143,A 122.3574,B 24.9502,C -1.6302,E1 24.9055,E2 684.0412} C_DIS
LIN {X -73.8226,Y 106.0075,Z 143,A 120.5339,B 24.9501,C -1.6325,E1 24.9097,E2 685.8653} C_DIS
LIN {X -70.3867,Y 108.3193,Z 143,A 118.6905,B 24.9499,C -1.6359,E1 24.914,E2 687.7069} C_DIS
LIN {X -66.9381,Y 110.4838,Z 143,A 116.8666,B 24.9497,C -1.6384,E1 24.9183,E2 689.5304} C_DIS
LIN {X -63.3674,Y 112.5698,Z 143,A 115.0347,B 24.9495,C -1.6419,E1 24.9227,E2 691.3596} C_DIS
LIN {X -59.6528,Y 114.5802,Z 143,A 113.2515,B 24.949,C -1.6494,E1 24.9271,E2 693.1299} C_DIS
LIN {X -56.6984,Y 116.0708,Z 143,A 111.7512,B 24.949,C -1.6502,E1 24.9308,E2 694.6321} C_DIS
LIN {X -53.9468,Y 117.3743,Z 143,A 110.3629,B 24.949,C -1.6506,E1 24.9344,E2 696.0231} C_DIS
LIN {X -50.5246,Y 118.8899,Z 143,A 108.7482,B 24.9487,C -1.6552,E1 24.9385,E2 697.6307} C_DIS
LIN {X -47.5506,Y 120.1103,Z 143,A 107.3196,B 24.9485,C -1.6571,E1 24.9422,E2 699.0579} C_DIS
LIN {X -44.5625,Y 121.2507,Z 143,A 105.8986,B 24.9485,C -1.6588,E1 24.9459,E2 700.4777} C_DIS
LIN {X -40.8005,Y 122.5652,Z 143,A 104.1196,B 24.9483,C -1.6605,E1 24.9506,E2 702.256} C_DIS
LIN {X -37.7067,Y 123.5521,Z 143,A 102.6833,B 24.9483,C -1.6624,E1 24.9544,E2 703.6904} C_DIS
LIN {X -34.6942,Y 124.4317,Z 143,A 101.2765,B 24.9482,C -1.6632,E1 24.9582,E2 705.0975} C_DIS
LIN {X -31.3616,Y 125.3139,Z 143,A 99.7445,B 24.9481,C -1.6646,E1 24.9623,E2 706.6285} C_DIS
LIN {X -28.4576,Y 126.0048,Z 143,A 98.4452,B 24.9479,C -1.667,E1 24.9659,E2 707.9238} C_DIS
LIN {X -25.625,Y 126.6109,Z 143,A 97.1162,B 24.9479,C -1.666,E1 24.9695,E2 709.2567} C_DIS
LIN {X -22.6078,Y 127.1844,Z 143,A 95.7428,B 24.9479,C -1.6665,E1 24.9733,E2 710.6302} C_DIS
LIN {X -19.4781,Y 127.7014,Z 143,A 94.377,B 24.9478,C -1.6695,E1 24.977,E2 711.9902} C_DIS
LIN {X -15.709,Y 128.22,Z 143,A 92.6183,B 24.9479,C -1.6671,E1 24.9819,E2 713.756} C_DIS
LIN {X -12.2493,Y 128.5961,Z 143,A 91.1556,B 24.9476,C -1.6719,E1 24.9859,E2 715.2082} C_DIS
LIN {X -8.9248,Y 128.8704,Z 143,A 89.6624,B 24.9476,C -1.6719,E1 24.9901,E2 716.7021} C_DIS
LIN {X -5.7589,Y 129.0518,Z 143,A 88.0981,B 24.9481,C -1.6646,E1 24.9945,E2 718.284} C_DIS
LIN {X -2.056,Y 129.1619,Z 143,A 86.601,B 24.9476,C -1.6723,E1 24.9986,E2 719.7631} C_DIS
LIN {X 1.8756,Y 129.1649,Z 143,A 84.8047,B 24.9477,C -1.67,E1 25.0037,E2 721.5647} C_DIS
LIN {X 5.7589,Y 129.0518,Z 143,A 83.1296,B 24.9476,C -1.6725,E1 25.0083,E2 723.2334} C_DIS
LIN {X 9.3107,Y 128.8422,Z 143,A 81.577,B 24.9476,C -1.6737,E1 25.0127,E2 724.7824} C_DIS
LIN {X 12.2493,Y 128.5961,Z 143,A 80.2285,B 24.9476,C -1.6716,E1 25.0164,E2 726.1352} C_DIS
LIN {X 15.2057,Y 128.2801,Z 143,A 78.9077,B 24.9476,C -1.6713,E1 25.0201,E2 727.4559} C_DIS
LIN {X 18.1778,Y 127.8927,Z 143,A 77.5763,B 24.9476,C -1.6708,E1 25.0238,E2 728.7871} C_DIS
LIN {X 21.3565,Y 127.4005,Z 143,A 76.1869,B 24.9476,C -1.6722,E1 25.0276,E2 730.1719} C_DIS
LIN {X 24.3533,Y 126.8617,Z 143,A 74.8162,B 24.9476,C -1.6707,E1 25.0313,E2 731.5447} C_DIS
LIN {X 27.6421,Y 126.1864,Z 143,A 73.3199,B 24.9478,C -1.6696,E1 25.0354,E2 733.0416} C_DIS
LIN {X 30.6436,Y 125.4913,Z 143,A 71.9531,B 24.9478,C -1.6688,E1 25.0391,E2 734.4084} C_DIS
LIN {X 33.6262,Y 124.725,Z 143,A 70.5853,B 24.9478,C -1.6678,E1 25.0428,E2 735.7764} C_DIS
LIN {X 36.6037,Y 123.8838,Z 143,A 69.2452,B 24.9478,C -1.6684,E1 25.0464,E2 737.1128} C_DIS
LIN {X 39.5851,Y 122.9635,Z 143,A 67.8541,B 24.9479,C -1.6669,E1 25.0501,E2 738.5048} C_DIS
LIN {X 42.8484,Y 121.8657,Z 143,A 66.3515,B 24.9479,C -1.6669,E1 25.0541,E2 740.0048} C_DIS
LIN {X 45.5669,Y 120.8744,Z 143,A 65.0449,B 24.9481,C -1.6644,E1 25.0575,E2 741.3142} C_DIS
LIN {X 48.576,Y 119.697,Z 143,A 63.6041,B 24.9482,C -1.6626,E1 25.0613,E2 742.7561} C_DIS
LIN {X 52.0055,Y 118.2496,Z 143,A 61.968,B 24.9482,C -1.6614,E1 25.0655,E2 744.3911} C_DIS
LIN {X 54.9527,Y 116.9091,Z 143,A 60.5341,B 24.9484,C -1.6598,E1 25.0691,E2 745.8251} C_DIS
LIN {X 57.7307,Y 115.5615,Z 143,A 59.1622,B 24.9484,C -1.658,E1 25.0725,E2 747.1978} C_DIS
LIN {X 60.3138,Y 114.2331,Z 143,A 57.917,B 24.9484,C -1.6585,E1 25.0756,E2 748.4383} C_DIS
LIN {X 63.6512,Y 112.4103,Z 143,A 56.0574,B 24.9492,C -1.6472,E1 25.0802,E2 750.3191} C_DIS
LIN {X 67.4339,Y 110.1819,Z 143,A 54.1562,B 24.9492,C -1.6466,E1 25.0847,E2 752.2158} C_DIS
LIN {X 71.2842,Y 107.7313,Z 143,A 52.1428,B 24.9494,C -1.6439,E1 25.0895,E2 754.2291} C_DIS
LIN {X 74.7264,Y 105.3729,Z 143,A 50.3018,B 24.9495,C -1.6412,E1 25.0937,E2 756.0701} C_DIS
LIN {X 78.0617,Y 102.9264,Z 143,A 48.4747,B 24.9497,C -1.6382,E1 25.0978,E2 757.8976} C_DIS
LIN {X 81.4221,Y 100.2895,Z 143,A 46.5988,B 24.9499,C -1.6356,E1 25.1019,E2 759.7727} C_DIS
LIN {X 84.6182,Y 97.6079,Z 143,A 44.7237,B 24.9502,C -1.6307,E1 25.1059,E2 761.6522} C_DIS
LIN {X 87.7296,Y 94.8212,Z 143,A 42.8992,B 24.9503,C -1.6283,E1 25.1096,E2 763.4748} C_DIS
LIN {X 90.6603,Y 92.0226,Z 143,A 41.094,B 24.9506,C -1.624,E1 25.1132,E2 765.2826} C_DIS
LIN {X 93.678,Y 88.9493,Z 143,A 39.2086,B 24.9508,C -1.6211,E1 25.1169,E2 767.1669} C_DIS
LIN {X 96.5056,Y 85.8732,Z 143,A 37.3646,B 24.951,C -1.6173,E1 25.1204,E2 769.0117} C_DIS
LIN {X 99.2297,Y 82.7104,Z 143,A 35.5025,B 24.9513,C -1.6123,E1 25.1237,E2 770.877} C_DIS
LIN {X 101.8465,Y 79.4659,Z 143,A 33.678,B 24.9515,C -1.609,E1 25.1269,E2 772.7007} C_DIS
LIN {X 104.3523,Y 76.1455,Z 143,A 31.7978,B 24.9519,C -1.6025,E1 25.13,E2 774.5871} C_DIS
LIN {X 106.8915,Y 72.5369,Z 143,A 29.9066,B 24.9519,C -1.6009,E1 25.133,E2 776.4729} C_DIS
LIN {X 109.211,Y 68.9951,Z 143,A 28.0438,B 24.9522,C -1.5967,E1 25.1358,E2 778.3363} C_DIS
LIN {X 111.5464,Y 65.1527,Z 143,A 26.0612,B 24.9525,C -1.5919,E1 25.1387,E2 780.3201} C_DIS
LIN {X 113.6017,Y 61.4996,Z 143,A 24.1889,B 24.9529,C -1.586,E1 25.1412,E2 782.1964} C_DIS
LIN {X 115.2706,Y 58.3068,Z 143,A 22.6726,B 24.9529,C -1.5858,E1 25.1431,E2 783.7052} C_DIS
LIN {X 116.7147,Y 55.3597,Z 143,A 21.2482,B 24.953,C -1.5833,E1 25.1449,E2 785.1279} C_DIS
LIN {X 118.2496,Y 52.0055,Z 143,A 19.6411,B 24.9532,C -1.58,E1 25.1467,E2 786.7341} C_DIS
LIN {X 119.341,Y 49.4443,Z 143,A 18.3894,B 24.9535,C -1.5755,E1 25.1481,E2 787.9895} C_DIS
LIN {X 120.5257,Y 46.4819,Z 143,A 17.014,B 24.9536,C -1.5734,E1 25.1495,E2 789.3623} C_DIS
LIN {X 121.6176,Y 43.5447,Z 143,A 15.6064,B 24.9539,C -1.5682,E1 25.1508,E2 790.7741} C_DIS
LIN {X 122.6316,Y 40.6011,Z 143,A 14.2557,B 24.9541,C -1.5656,E1 25.152,E2 792.1234} C_DIS
LIN {X 123.7527,Y 37.0513,Z 143,A 12.6228,B 24.9543,C -1.5614,E1 25.1534,E2 793.7568} C_DIS
LIN {X 124.4317,Y 34.6942,Z 143,A 11.5437,B 24.9545,C -1.5585,E1 25.1542,E2 794.8365} C_DIS
LIN {X 125.1835,Y 31.8753,Z 143,A 10.2602,B 24.9547,C -1.5551,E1 25.1551,E2 796.1208} C_DIS
LIN {X 125.9082,Y 28.8805,Z 143,A 8.8877,B 24.955,C -1.5504,E1 25.156,E2 797.4963} C_DIS
LIN {X 126.6004,Y 25.677,Z 143,A 7.4425,B 24.9552,C -1.5462,E1 25.1568,E2 798.943} C_DIS
LIN {X 127.2137,Y 22.4443,Z 143,A 6.0075,B 24.9554,C -1.5429,E1 25.1575,E2 800.3776} C_DIS
LIN {X 127.7372,Y 19.247,Z 143,A 4.6074,B 24.9556,C -1.5402,E1 25.1581,E2 801.7757} C_DIS
LIN {X 128.1802,Y 16.0428,Z 143,A 3.0003,B 24.9564,C -1.5263,E1 25.1587,E2 803.406} C_DIS
LIN {X 128.5961,Y 12.2493,Z 143,A 1.4905,B 24.9561,C -1.5306,E1 25.1591,E2 804.8968} C_DIS
LIN {X 128.8422,Y 9.3107,Z 143,A 0.1678,B 24.9564,C -1.5255,E1 25.1594,E2 806.2236} C_DIS
LIN {X 129.0518,Y 5.7589,Z 143,A -1.543,B 24.9571,C -1.5132,E1 25.1597,E2 807.9532} C_DIS
LIN {X 129.1618,Y 2.0656,Z 143,A -2.9891,B 24.9568,C -1.5182,E1 25.1597,E2 809.3791} C_DIS
LIN {X 129.1506,Y -2.7355,Z 143,A -5.2678,B 24.9577,C -1.5031,E1 25.1597,E2 811.6797} C_DIS
LIN {X 129.0105,Y -6.58,Z 143,A -6.8859,B 24.9577,C -1.5022,E1 25.1595,E2 813.2902} C_DIS
LIN {X 128.7819,Y -10.1378,Z 143,A -8.3827,B 24.9577,C -1.5015,E1 25.1592,E2 814.7799} C_DIS
LIN {X 128.4846,Y -13.3754,Z 143,A -9.9092,B 24.9583,C -1.4922,E1 25.1588,E2 816.3192} C_DIS
LIN {X 128.0702,Y -16.8821,Z 143,A -11.3381,B 24.9582,C -1.4944,E1 25.1583,E2 817.7345} C_DIS
LIN {X 127.642,Y -19.8619,Z 143,A -12.7046,B 24.9585,C -1.4883,E1 25.1578,E2 819.1073} C_DIS
LIN {X 127.1665,Y -22.7079,Z 143,A -14.0061,B 24.9588,C -1.483,E1 25.1571,E2 820.4137} C_DIS
LIN {X 126.5642,Y -25.8549,Z 143,A -15.3915,B 24.959,C -1.4802,E1 25.1564,E2 821.7975} C_DIS
LIN {X 125.9122,Y -28.863,Z 143,A -16.7493,B 24.9592,C -1.4762,E1 25.1556,E2 823.157} C_DIS
LIN {X 125.1579,Y -31.9763,Z 143,A -18.196,B 24.9595,C -1.4702,E1 25.1546,E2 824.6096} C_DIS
LIN {X 124.2943,Y -35.1856,Z 143,A -19.6265,B 24.9596,C -1.4677,E1 25.1535,E2 826.0376} C_DIS
LIN {X 123.4277,Y -38.1133,Z 143,A -20.9647,B 24.9598,C -1.4642,E1 25.1524,E2 827.3764} C_DIS
LIN {X 122.3537,Y -41.4358,Z 143,A -22.5197,B 24.9601,C -1.4589,E1 25.1511,E2 828.9352} C_DIS
LIN {X 120.9174,Y -45.4523,Z 143,A -24.3997,B 24.9604,C -1.4535,E1 25.1493,E2 830.8172} C_DIS
LIN {X 119.7395,Y -48.4706,Z 143,A -25.8366,B 24.9607,C -1.449,E1 25.1478,E2 832.2568} C_DIS
LIN {X 118.41,Y -51.6346,Z 143,A -27.3616,B 24.9609,C -1.4441,E1 25.1461,E2 833.7851} C_DIS
LIN {X 116.9091,Y -54.9527,Z 143,A -28.9465,B 24.9611,C -1.4407,E1 25.1443,E2 835.3694} C_DIS
LIN {X 115.6119,Y -57.6285,Z 143,A -30.2559,B 24.9613,C -1.4372,E1 25.1427,E2 836.68} C_DIS
LIN {X 114.1793,Y -60.4164,Z 143,A -31.6506,B 24.9615,C -1.4328,E1 25.1409,E2 838.0778} C_DIS
LIN {X 112.3522,Y -63.753,Z 143,A -33.451,B 24.9621,C -1.4217,E1 25.1384,E2 839.8949} C_DIS
LIN {X 110.1393,Y -67.5034,Z 143,A -35.3162,B 24.9623,C -1.4195,E1 25.1357,E2 841.7557} C_DIS
LIN {X 107.8664,Y -71.0789,Z 143,A -37.1634,B 24.9625,C -1.4158,E1 25.1329,E2 843.6025} C_DIS
LIN {X 105.593,Y -74.4143,Z 143,A -38.9661,B 24.9628,C -1.41,E1 25.13,E2 845.4099} C_DIS
LIN {X 102.9691,Y -78.0051,Z 143,A -40.9428,B 24.9631,C -1.4043,E1 25.1267,E2 847.3905} C_DIS
LIN {X 100.3001,Y -81.4089,Z 143,A -42.8328,B 24.9633,C -1.4006,E1 25.1234,E2 849.2805} C_DIS
LIN {X 97.6079,Y -84.6182,Z 143,A -44.7162,B 24.9636,C -1.3943,E1 25.12,E2 851.1701} C_DIS
LIN {X 94.8212,Y -87.7296,Z 143,A -46.5386,B 24.9638,C -1.3911,E1 25.1166,E2 852.9921} C_DIS
LIN {X 91.9335,Y -90.7511,Z 143,A -48.3827,B 24.964,C -1.3869,E1 25.113,E2 854.838} C_DIS
LIN {X 88.919,Y -93.7065,Z 143,A -50.2908,B 24.9643,C -1.3805,E1 25.1092,E2 856.7536} C_DIS
LIN {X 85.7038,Y -96.6554,Z 143,A -52.1903,B 24.9644,C -1.3777,E1 25.1052,E2 858.6519} C_DIS
LIN {X 82.3476,Y -99.5301,Z 143,A -54.1119,B 24.9646,C -1.3753,E1 25.1011,E2 860.5719} C_DIS
LIN {X 78.8491,Y -102.3246,Z 143,A -56.0628,B 24.9647,C -1.3727,E1 25.0968,E2 862.5216} C_DIS
LIN {X 75.4727,Y -104.8399,Z 143,A -58.0065,B 24.9651,C -1.3647,E1 25.0924,E2 864.4773} C_DIS
LIN {X 71.9621,Y -107.2796,Z 143,A -59.8742,B 24.9652,C -1.3623,E1 25.0881,E2 866.3443} C_DIS
LIN {X 68.2958,Y -109.6497,Z 143,A -61.7491,B 24.9652,C -1.3617,E1 25.0837,E2 868.2145} C_DIS
LIN {X 64.6742,Y -111.824,Z 143,A -63.5998,B 24.9654,C -1.3594,E1 25.0793,E2 870.065} C_DIS
LIN {X 61.0926,Y -113.8203,Z 143,A -65.4101,B 24.9655,C -1.3566,E1 25.0748,E2 871.8767} C_DIS
LIN {X 57.8782,Y -115.4888,Z 143,A -66.955,B 24.9655,C -1.357,E1 25.071,E2 873.4164} C_DIS
LIN {X 55.254,Y -116.7651,Z 143,A -68.2633,B 24.9657,C -1.3542,E1 25.0677,E2 874.7279} C_DIS
LIN {X 52.3737,Y -118.0849,Z 143,A -69.6746,B 24.9657,C -1.3517,E1 25.0641,E2 876.1416} C_DIS
LIN {X 48.0933,Y -119.8915,Z 143,A -71.7238,B 24.9659,C -1.3492,E1 25.0588,E2 878.1918} C_DIS
LIN {X 44.9096,Y -121.1207,Z 143,A -73.165,B 24.9659,C -1.3509,E1 25.0551,E2 879.6261} C_DIS
LIN {X 42.2169,Y -122.0846,Z 143,A -74.4658,B 24.9659,C -1.3476,E1 25.0516,E2 880.9321} C_DIS
LIN {X 39.2117,Y -123.0828,Z 143,A -75.8762,B 24.9661,C -1.3455,E1 25.0479,E2 882.3446} C_DIS
LIN {X 35.9177,Y -124.0846,Z 143,A -77.3875,B 24.9661,C -1.3445,E1 25.0438,E2 883.8556} C_DIS
LIN {X 32.9588,Y -124.903,Z 143,A -78.7714,B 24.9663,C -1.3419,E1 25.0401,E2 885.2435} C_DIS
LIN {X 30.1396,Y -125.6127,Z 143,A -80.0516,B 24.9663,C -1.3411,E1 25.0366,E2 886.5238} C_DIS
LIN {X 26.9306,Y -126.34,Z 143,A -81.4821,B 24.9663,C -1.3412,E1 25.0327,E2 887.9521} C_DIS
LIN {X 23.5564,Y -127.014,Z 143,A -83.1661,B 24.9668,C -1.3318,E1 25.0281,E2 889.6563} C_DIS
LIN {X 19.8623,Y -127.642,Z 143,A -84.6978,B 24.9665,C -1.3372,E1 25.0239,E2 891.1738} C_DIS
LIN {X 16.8821,Y -128.0702,Z 143,A -86.0287,B 24.9665,C -1.3366,E1 25.0202,E2 892.5051} C_DIS
LIN {X 13.2745,Y -128.4954,Z 143,A -87.7422,B 24.9668,C -1.3304,E1 25.0154,E2 894.2321} C_DIS
LIN {X 9.4455,Y -128.8324,Z 143,A -89.3289,B 24.9666,C -1.3355,E1 25.011,E2 895.8057} C_DIS
LIN {X 5.7589,Y -129.0518,Z 143,A -91.1039,B 24.967,C -1.3279,E1 25.006,E2 897.5982} C_DIS
LIN {X 2.056,Y -129.1619,Z 143,A -92.6437,B 24.9667,C -1.3327,E1 25.0017,E2 899.1265} C_DIS
LIN {X 2.056,Y -129.1619,Z 143,A -92.6437,B 24.9667,C -1.3327,E1 25.0017,E2 899.1265} C_DIS
Enddeposition()
LIN {X 0.9147,Y -128.1906,Z 143,A -93.102,B 24.8918,C -1.3367,E1 24.9259,E2 899.5652} C_DIS
Startdeposition()
$VEL.CP = VEL_PRINT
LIN {X 4.1973,Y -128.1453,Z 143,A -90.5109,B 24.8889,C -1.3935,E1 24.9335,E2 896.8397} C_DIS
LIN {X 8.2432,Y -127.9477,Z 143,A -89.1721,B 24.8901,C -1.3702,E1 24.9371,E2 895.5565} C_DIS
LIN {X 11.0813,Y -127.733,Z 143,A -87.1583,B 24.8881,C -1.4088,E1 24.943,E2 893.4523} C_DIS
LIN {X 16.5291,Y -127.1425,Z 143,A -85.6463,B 24.8905,C -1.3624,E1 24.9468,E2 892.0516} C_DIS
LIN {X 19.5607,Y -126.7114,Z 143,A -84.0989,B 24.89,C -1.3725,E1 24.9511,E2 890.4817} C_DIS
LIN {X 23.3792,Y -126.0647,Z 143,A -82.268,B 24.8896,C -1.379,E1 24.9562,E2 888.6375} C_DIS
LIN {X 27.17,Y -125.3003,Z 143,A -80.6852,B 24.8899,C -1.3731,E1 24.9605,E2 887.0705} C_DIS
LIN {X 30.3984,Y -124.5569,Z 143,A -79.0487,B 24.8894,C -1.3826,E1 24.965,E2 885.4139} C_DIS
LIN {X 34.4406,Y -123.4998,Z 143,A -77.2716,B 24.8896,C -1.38,E1 24.9698,E2 883.6458} C_DIS
LIN {X 37.6925,Y -122.5465,Z 143,A -75.4421,B 24.8886,C -1.3981,E1 24.9748,E2 881.7768} C_DIS
LIN {X 41.1125,Y -121.4434,Z 143,A -74.2237,B 24.8896,C -1.38,E1 24.9779,E2 880.6035} C_DIS
LIN {X 44.5731,Y -120.2154,Z 143,A -72.4969,B 24.8892,C -1.3867,E1 24.9824,E2 878.8645} C_DIS
LIN {X 48.0311,Y -118.8753,Z 143,A -70.5973,B 24.8884,C -1.4016,E1 24.9874,E2 876.9337} C_DIS
LIN {X 51.0445,Y -117.6129,Z 143,A -69.4922,B 24.8893,C -1.3854,E1 24.9902,E2 875.8698} C_DIS
LIN {X 54.0748,Y -116.251,Z 143,A -68.0095,B 24.8892,C -1.3876,E1 24.9939,E2 874.3855} C_DIS
LIN {X 57.0263,Y -114.8322,Z 143,A -66.1475,B 24.888,C -1.4108,E1 24.9987,E2 872.4735} C_DIS
LIN {X 60.2447,Y -113.178,Z 143,A -64.5834,B 24.888,C -1.4108,E1 25.0026,E2 870.9138} C_DIS
LIN {X 63.176,Y -111.5688,Z 143,A -63.2806,B 24.8883,C -1.4036,E1 25.0057,E2 869.6322} C_DIS
LIN {X 67.2358,Y -109.1705,Z 143,A -61.0777,B 24.8879,C -1.4126,E1 25.011,E2 867.4147} C_DIS
LIN {X 70.1582,Y -107.3163,Z 143,A -59.6851,B 24.8881,C -1.4075,E1 25.0142,E2 866.0386} C_DIS
LIN {X 73.6559,Y -104.9461,Z 143,A -57.7882,B 24.8879,C -1.4119,E1 25.0186,E2 864.1379} C_DIS
LIN {X 77.2334,Y -102.3415,Z 143,A -55.7334,B 24.8875,C -1.4202,E1 25.0232,E2 862.0709} C_DIS
LIN {X 81.0173,Y -99.3731,Z 143,A -53.7453,B 24.8877,C -1.4165,E1 25.0275,E2 860.099} C_DIS
LIN {X 84.1041,Y -96.7748,Z 143,A -51.9167,B 24.8874,C -1.4221,E1 25.0314,E2 858.2644} C_DIS
LIN {X 87.2198,Y -93.9763,Z 143,A -49.9992,B 24.887,C -1.429,E1 25.0354,E2 856.3383} C_DIS
LIN {X 90.1032,Y -91.2159,Z 143,A -48.2578,B 24.8869,C -1.4311,E1 25.0388,E2 854.5992} C_DIS
LIN {X 93.1307,Y -88.122,Z 143,A -46.354,B 24.8867,C -1.4344,E1 25.0425,E2 852.6959} C_DIS
LIN {X 96.0151,Y -84.9699,Z 143,A -44.3661,B 24.8862,C -1.4435,E1 25.0463,E2 850.6952} C_DIS
LIN {X 99.58,Y -80.7635,Z 143,A -42.1354,B 24.8865,C -1.4377,E1 25.0502,E2 848.4885} C_DIS
LIN {X 101.6517,Y -78.1397,Z 143,A -40.4849,B 24.8858,C -1.4501,E1 25.0531,E2 846.8165} C_DIS
LIN {X 104.2974,Y -74.571,Z 143,A -38.539,B 24.8857,C -1.4536,E1 25.0563,E2 844.8719} C_DIS
LIN {X 106.6403,Y -71.1804,Z 143,A -36.2844,B 24.8841,C -1.481,E1 25.0599,E2 842.5637} C_DIS
LIN {X 108.9552,Y -67.5839,Z 143,A -35.1035,B 24.886,C -1.4475,E1 25.0615,E2 841.468} C_DIS
LIN {X 111.5448,Y -63.2193,Z 143,A -32.5204,B 24.8847,C -1.471,E1 25.0652,E2 838.8428} C_DIS
LIN {X 113.4965,Y -59.6393,Z 143,A -30.8267,B 24.8847,C -1.4696,E1 25.0674,E2 837.1611} C_DIS
LIN {X 114.9448,Y -56.798,Z 143,A -29.4324,B 24.8847,C -1.4723,E1 25.0692,E2 835.7679} C_DIS
LIN {X 118.3765,Y -49.248,Z 143,A -25.7217,B 24.884,C -1.484,E1 25.0734,E2 832.05} C_DIS
LIN {X 119.8532,Y -45.5403,Z 143,A -23.4972,B 24.8823,C -1.5132,E1 25.0757,E2 829.7687} C_DIS
LIN {X 121.1968,Y -41.8294,Z 143,A -22.227,B 24.8835,C -1.4924,E1 25.0768,E2 828.555} C_DIS
LIN {X 122.2321,Y -38.701,Z 143,A -20.6538,B 24.8829,C -1.5025,E1 25.0782,E2 826.9668} C_DIS
LIN {X 123.3906,Y -34.8312,Z 143,A -18.8963,B 24.8827,C -1.5057,E1 25.0795,E2 825.2118} C_DIS
LIN {X 124.3309,Y -31.3089,Z 143,A -17.3468,B 24.8827,C -1.5067,E1 25.0806,E2 823.6688} C_DIS
LIN {X 125.1723,Y -27.7631,Z 143,A -15.5305,B 24.8818,C -1.5221,E1 25.0817,E2 821.8268} C_DIS
LIN {X 126.0174,Y -23.6262,Z 143,A -13.7202,B 24.8817,C -1.5242,E1 25.0827,E2 820.0222} C_DIS
LIN {X 126.9486,Y -17.9579,Z 143,A -11.0219,B 24.8808,C -1.5397,E1 25.0838,E2 817.3032} C_DIS
LIN {X 127.5398,Y -13.1295,Z 143,A -9.1138,B 24.8812,C -1.5326,E1 25.0844,E2 815.4233} C_DIS
LIN {X 127.861,Y -9.488,Z 143,A -7.0076,B 24.8794,C -1.5634,E1 25.0849,E2 813.2567} C_DIS
LIN {X 128.1056,Y -5.2406,Z 143,A -4.8169,B 24.8781,C -1.5853,E1 25.0851,E2 811.0273} C_DIS
LIN {X 128.2131,Y 0.6098,Z 143,A -3.2003,B 24.8808,C -1.5402,E1 25.0851,E2 809.527} C_DIS
LIN {X 127.9871,Y 7.6038,Z 143,A -0.1464,B 24.8804,C -1.5464,E1 25.0849,E2 806.4764} C_DIS
LIN {X 127.6369,Y 12.1352,Z 143,A 2.1029,B 24.8793,C -1.5647,E1 25.0843,E2 804.1974} C_DIS
LIN {X 127.21,Y 16.0138,Z 143,A 3.9195,B 24.8788,C -1.5742,E1 25.0837,E2 802.3691} C_DIS
LIN {X 126.6995,Y 19.6373,Z 143,A 5.477,B 24.8788,C -1.5754,E1 25.0831,E2 800.818} C_DIS
LIN {X 126.0918,Y 23.2308,Z 143,A 7.1787,B 24.8782,C -1.5845,E1 25.0823,E2 799.1048} C_DIS
LIN {X 125.3365,Y 27.0026,Z 143,A 8.7612,B 24.8782,C -1.5827,E1 25.0814,E2 797.5358} C_DIS
LIN {X 124.5974,Y 30.2305,Z 143,A 10.2122,B 24.8781,C -1.5858,E1 25.0804,E2 796.0859} C_DIS
LIN {X 123.7908,Y 33.3815,Z 143,A 11.7392,B 24.8776,C -1.5943,E1 25.0793,E2 794.5477} C_DIS
LIN {X 121.9229,Y 39.6687,Z 143,A 14.5427,B 24.8774,C -1.5965,E1 25.0771,E2 791.7549} C_DIS
LIN {X 120.5686,Y 43.6068,Z 143,A 16.4372,B 24.877,C -1.604,E1 25.0753,E2 789.8535} C_DIS
LIN {X 119.2056,Y 47.2117,Z 143,A 18.477,B 24.8757,C -1.626,E1 25.0732,E2 787.7731} C_DIS
LIN {X 117.9702,Y 50.2182,Z 143,A 19.558,B 24.8766,C -1.6105,E1 25.0721,E2 786.7345} C_DIS
LIN {X 116.2663,Y 54.0417,Z 143,A 21.4455,B 24.8762,C -1.6169,E1 25.0699,E2 784.8422} C_DIS
LIN {X 114.8183,Y 57.0544,Z 143,A 22.8304,B 24.8763,C -1.6154,E1 25.0682,E2 783.4682} C_DIS
LIN {X 113.6147,Y 59.4142,Z 143,A 24.1136,B 24.8758,C -1.624,E1 25.0665,E2 782.1715} C_DIS
LIN {X 111.601,Y 63.12,Z 143,A 26.093,B 24.8752,C -1.6342,E1 25.0638,E2 780.1784} C_DIS
LIN {X 109.2849,Y 67.0493,Z 143,A 28.0819,B 24.875,C -1.6372,E1 25.061,E2 778.1928} C_DIS
LIN {X 106.9171,Y 70.7646,Z 143,A 30.0399,B 24.8747,C -1.6418,E1 25.058,E2 776.2336} C_DIS
LIN {X 104.5469,Y 74.2218,Z 143,A 31.9502,B 24.8743,C -1.6486,E1 25.055,E2 774.3167} C_DIS
LIN {X 102.0248,Y 77.6519,Z 143,A 33.8472,B 24.874,C -1.6531,E1 25.0518,E2 772.4182} C_DIS
LIN {X 98.9895,Y 81.4862,Z 143,A 36.0211,B 24.8737,C -1.6578,E1 25.048,E2 770.2432} C_DIS
LIN {X 96.2345,Y 84.7218,Z 143,A 37.9155,B 24.8734,C -1.662,E1 25.0445,E2 768.3474} C_DIS
LIN {X 93.2033,Y 88.0451,Z 143,A 39.8783,B 24.8733,C -1.6641,E1 25.0408,E2 766.3882} C_DIS
LIN {X 90.1257,Y 91.1935,Z 143,A 41.8719,B 24.8729,C -1.6698,E1 25.0368,E2 764.3898} C_DIS
LIN {X 87.023,Y 94.1589,Z 143,A 43.8042,B 24.8726,C -1.6746,E1 25.0329,E2 762.4541} C_DIS
LIN {X 83.6472,Y 97.1696,Z 143,A 45.7508,B 24.8726,C -1.6748,E1 25.0288,E2 760.5147} C_DIS
LIN {X 80.4546,Y 99.8291,Z 143,A 47.6144,B 24.8724,C -1.6787,E1 25.0248,E2 758.649} C_DIS
LIN {X 76.9266,Y 102.5731,Z 143,A 49.5877,B 24.8722,C -1.6811,E1 25.0204,E2 756.6771} C_DIS
LIN {X 73.5451,Y 105.024,Z 143,A 51.5325,B 24.8718,C -1.6884,E1 25.016,E2 754.7217} C_DIS
LIN {X 69.7386,Y 107.5887,Z 143,A 53.5204,B 24.8718,C -1.6886,E1 25.0113,E2 752.7402} C_DIS
LIN {X 66.0163,Y 109.9126,Z 143,A 55.3582,B 24.872,C -1.6853,E1 25.007,E2 750.916} C_DIS
LIN {X 62.8398,Y 111.7584,Z 143,A 57.0886,B 24.8715,C -1.6922,E1 25.0028,E2 749.1743} C_DIS
LIN {X 59.384,Y 113.6306,Z 143,A 58.8067,B 24.8715,C -1.6927,E1 24.9986,E2 747.46} C_DIS
LIN {X 55.1609,Y 115.7393,Z 143,A 60.8596,B 24.8715,C -1.6925,E1 24.9934,E2 745.413} C_DIS
LIN {X 52.1653,Y 117.1202,Z 143,A 62.3356,B 24.8714,C -1.6943,E1 24.9897,E2 743.9364} C_DIS
LIN {X 47.8301,Y 118.9563,Z 143,A 64.398,B 24.8714,C -1.6945,E1 24.9844,E2 741.8784} C_DIS
LIN {X 44.946,Y 120.0757,Z 143,A 65.8117,B 24.8712,C -1.6974,E1 24.9807,E2 740.4609} C_DIS
LIN {X 41.5839,Y 121.2819,Z 143,A 67.6793,B 24.8702,C -1.7126,E1 24.9757,E2 738.561} C_DIS
LIN {X 37.1183,Y 122.7223,Z 143,A 69.6349,B 24.8706,C -1.7071,E1 24.9705,E2 736.622} C_DIS
LIN {X 33.1462,Y 123.8535,Z 143,A 71.3642,B 24.8709,C -1.7025,E1 24.9659,E2 734.9064} C_DIS
LIN {X 29.8499,Y 124.6892,Z 143,A 72.8739,B 24.8709,C -1.7029,E1 24.9618,E2 733.3979} C_DIS
LIN {X 26.0231,Y 125.5444,Z 143,A 74.7061,B 24.8705,C -1.7078,E1 24.9567,E2 731.5566} C_DIS
LIN {X 22.2934,Y 126.2596,Z 143,A 76.4072,B 24.8705,C -1.7087,E1 24.9521,E2 729.8553} C_DIS
LIN {X 18.2161,Y 126.9117,Z 143,A 78.2317,B 24.8705,C -1.7082,E1 24.947,E2 728.0337} C_DIS
LIN {X 14.1278,Y 127.4323,Z 143,A 80.0499,B 24.8705,C -1.7073,E1 24.942,E2 726.2188} C_DIS
LIN {X 10.5686,Y 127.7763,Z 143,A 82.0252,B 24.8693,C -1.7263,E1 24.9364,E2 724.1996} C_DIS
LIN {X 6.7471,Y 128.0352,Z 143,A 83.2787,B 24.8708,C -1.7035,E1 24.9331,E2 723.0007} C_DIS
LIN {X -0.7111,Y 128.2106,Z 143,A 86.6511,B 24.8708,C -1.7049,E1 24.9236,E2 719.6256} C_DIS
LIN {X -9.6299,Y 127.8506,Z 143,A 90.5536,B 24.8711,C -1.6991,E1 24.9128,E2 715.7357} C_DIS
LIN {X -12.6208,Y 127.5902,Z 143,A 91.9762,B 24.8709,C -1.7024,E1 24.9088,E2 714.3046} C_DIS
LIN {X -16.5225,Y 127.1433,Z 143,A 93.7824,B 24.8708,C -1.7039,E1 24.9038,E2 712.4937} C_DIS
LIN {X -20.6796,Y 126.5343,Z 143,A 95.6751,B 24.8708,C -1.7033,E1 24.8986,E2 710.6007} C_DIS
LIN {X -24.1833,Y 125.9109,Z 143,A 97.2251,B 24.871,C -1.7001,E1 24.8943,E2 709.0567} C_DIS
LIN {X -28.0264,Y 125.1127,Z 143,A 98.875,B 24.8714,C -1.6935,E1 24.8898,E2 707.4205} C_DIS
LIN {X -31.365,Y 124.3166,Z 143,A 100.5242,B 24.8712,C -1.6976,E1 24.8853,E2 705.7593} C_DIS
LIN {X -34.6662,Y 123.4367,Z 143,A 102.0445,B 24.8713,C -1.6957,E1 24.8813,E2 704.2411} C_DIS
LIN {X -39.19,Y 122.0759,Z 143,A 104.1994,B 24.8713,C -1.6953,E1 24.8755,E2 702.0833} C_DIS
LIN {X -45.3117,Y 119.9388,Z 143,A 107.2751,B 24.871,C -1.7001,E1 24.8674,E2 698.99} C_DIS
LIN {X -48.6292,Y 118.6342,Z 143,A 108.814,B 24.8713,C -1.6952,E1 24.8634,E2 697.4594} C_DIS
LIN {X -52.4992,Y 116.9708,Z 143,A 110.5521,B 24.8719,C -1.6855,E1 24.859,E2 695.7403} C_DIS
LIN {X -55.4243,Y 115.6135,Z 143,A 111.9881,B 24.8721,C -1.683,E1 24.8554,E2 694.3066} C_DIS
LIN {X -58.4076,Y 114.1356,Z 143,A 113.5075,B 24.8721,C -1.682,E1 24.8516,E2 692.7855} C_DIS
LIN {X -61.8106,Y 112.3315,Z 143,A 115.3403,B 24.8721,C -1.6843,E1 24.8471,E2 690.942} C_DIS
LIN {X -65.9314,Y 109.9634,Z 143,A 117.36,B 24.8726,C -1.6755,E1 24.8422,E2 688.9373} C_DIS
LIN {X -69.1535,Y 107.9657,Z 143,A 119.1793,B 24.8724,C -1.6782,E1 24.8379,E2 687.1058} C_DIS
LIN {X -72.3661,Y 105.8395,Z 143,A 120.8916,B 24.8727,C -1.6743,E1 24.834,E2 685.397} C_DIS
LIN {X -76.045,Y 103.2278,Z 143,A 122.8564,B 24.8731,C -1.6676,E1 24.8295,E2 683.4412} C_DIS
LIN {X -79.1981,Y 100.8288,Z 143,A 125.0878,B 24.8719,C -1.6856,E1 24.8245,E2 681.1586} C_DIS
LIN {X -82.4697,Y 98.171,Z 143,A 127.2454,B 24.8714,C -1.6944,E1 24.8199,E2 678.9717} C_DIS
LIN {X -86.6317,Y 94.5186,Z 143,A 128.8266,B 24.8744,C -1.6463,E1 24.8168,E2 677.4989} C_DIS
LIN {X -89.9603,Y 91.3552,Z 143,A 131.2037,B 24.8738,C -1.6566,E1 24.812,E2 675.0874} C_DIS
LIN {X -93.6757,Y 87.5414,Z 143,A 133.6987,B 24.8738,C -1.656,E1 24.8071,E2 672.5829} C_DIS
LIN {X -97.0803,Y 83.7509,Z 143,A 136.3968,B 24.8729,C -1.6699,E1 24.8021,E2 669.8393} C_DIS
LIN {X -100.3512,Y 79.8024,Z 143,A 138.047,B 24.8752,C -1.6336,E1 24.7994,E2 668.268} C_DIS
LIN {X -102.7902,Y 76.6353,Z 143,A 139.9034,B 24.8752,C -1.632,E1 24.7962,E2 666.4066} C_DIS
LIN {X -105.46,Y 72.9185,Z 143,A 141.9877,B 24.8755,C -1.6281,E1 24.7929,E2 664.3214} C_DIS
LIN {X -107.8919,Y 69.2688,Z 143,A 143.9413,B 24.8759,C -1.6222,E1 24.7899,E2 662.372} C_DIS
LIN {X -110.1824,Y 65.5641,Z 143,A 146.0266,B 24.8759,C -1.623,E1 24.7869,E2 660.2741} C_DIS
LIN {X -112.7187,Y 61.1015,Z 143,A 148.2006,B 24.8766,C -1.6106,E1 24.7839,E2 658.1182} C_DIS
LIN {X -114.3777,Y 57.932,Z 143,A 149.6867,B 24.8772,C -1.6006,E1 24.7821,E2 656.648} C_DIS
LIN {X -115.8153,Y 55.0019,Z 143,A 151.1861,B 24.8774,C -1.598,E1 24.7802,E2 655.1466} C_DIS
LIN {X -117.26,Y 51.8526,Z 143,A 152.9256,B 24.8771,C -1.6021,E1 24.7782,E2 653.3878} C_DIS
LIN {X -118.9326,Y 47.8891,Z 143,A 154.6635,B 24.878,C -1.5876,E1 24.7764,E2 651.6749} C_DIS
LIN {X -120.1484,Y 44.752,Z 143,A 156.2182,B 24.8781,C -1.5852,E1 24.7749,E2 650.1171} C_DIS
LIN {X -121.2552,Y 41.661,Z 143,A 157.6745,B 24.8784,C -1.5801,E1 24.7735,E2 648.6648} C_DIS
LIN {X -123.1739,Y 35.5913,Z 143,A 160.4872,B 24.8791,C -1.5694,E1 24.7712,E2 645.8613} C_DIS
LIN {X -124.0281,Y 32.4917,Z 143,A 162.2695,B 24.8784,C -1.5808,E1 24.7699,E2 644.0414} C_DIS
LIN {X -125.1503,Y 27.8615,Z 143,A 164.0827,B 24.8797,C -1.5592,E1 24.7688,E2 642.269} C_DIS
LIN {X -125.8622,Y 24.4381,Z 143,A 165.7642,B 24.8797,C -1.5596,E1 24.7679,E2 640.5766} C_DIS
LIN {X -126.5419,Y 20.6337,Z 143,A 167.4097,B 24.8802,C -1.5502,E1 24.7671,E2 638.9438} C_DIS
LIN {X -127.0516,Y 17.2223,Z 143,A 169.0855,B 24.8802,C -1.5514,E1 24.7664,E2 637.2553} C_DIS
LIN {X -127.4903,Y 13.5886,Z 143,A 170.6165,B 24.8807,C -1.5412,E1 24.766,E2 635.7394} C_DIS
LIN {X -127.8493,Y 9.6476,Z 143,A 172.467,B 24.8808,C -1.5391,E1 24.7655,E2 633.8827} C_DIS
LIN {X -128.0799,Y 5.857,Z 143,A 174.2015,B 24.8811,C -1.5352,E1 24.7653,E2 632.147} C_DIS
LIN {X -128.1963,Y 2.0423,Z 143,A 175.8671,B 24.8815,C -1.5278,E1 24.7652,E2 630.489} C_DIS
LIN {X -128.1864,Y -2.6329,Z 143,A 178.06,B 24.8816,C -1.5257,E1 24.7652,E2 628.2879} C_DIS
LIN {X -128.0379,Y -6.6937,Z 143,A 179.8798,B 24.8819,C -1.52,E1 24.7655,E2 626.4709} C_DIS
LIN {X -127.7602,Y -10.7592,Z 143,A -178.3853,B 24.8825,C -1.5101,E1 24.7658,E2 624.7492} C_DIS
LIN {X -127.3611,Y -14.756,Z 143,A -176.5317,B 24.8827,C -1.5069,E1 24.7664,E2 622.8919} C_DIS
LIN {X -126.911,Y -18.2208,Z 143,A -174.9439,B 24.8829,C -1.5031,E1 24.767,E2 621.3037} C_DIS
LIN {X -126.2287,Y -22.4658,Z 143,A -173.0365,B 24.8833,C -1.4963,E1 24.7679,E2 619.4012} C_DIS
LIN {X -125.2228,Y -27.5293,Z 143,A -170.7992,B 24.8839,C -1.4857,E1 24.7691,E2 617.176} C_DIS
LIN {X -124.433,Y -30.9065,Z 143,A -169.065,B 24.8837,C -1.4894,E1 24.7703,E2 615.4227} C_DIS
LIN {X -123.3652,Y -34.9218,Z 143,A -167.3252,B 24.8843,C -1.4782,E1 24.7715,E2 613.6996} C_DIS
LIN {X -121.7856,Y -40.085,Z 143,A -165.0582,B 24.8851,C -1.464,E1 24.7734,E2 611.4535} C_DIS
LIN {X -120.625,Y -43.4503,Z 143,A -163.2695,B 24.8848,C -1.4684,E1 24.7751,E2 609.6441} C_DIS
LIN {X -119.4564,Y -46.5673,Z 143,A -161.8128,B 24.8852,C -1.4625,E1 24.7765,E2 608.1933} C_DIS
LIN {X -118.2421,Y -49.5696,Z 143,A -160.3829,B 24.8854,C -1.4574,E1 24.7781,E2 606.7676} C_DIS
LIN {X -117.0519,Y -52.318,Z 143,A -158.9878,B 24.8855,C -1.4562,E1 24.7796,E2 605.3677} C_DIS
LIN {X -113.9108,Y -58.8491,Z 143,A -155.3716,B 24.885,C -1.4646,E1 24.7842,E2 601.7119} C_DIS
LIN {X -112.266,Y -61.9289,Z 143,A -154.3105,B 24.8866,C -1.4368,E1 24.7855,E2 600.7116} C_DIS
LIN {X -110.7208,Y -64.6515,Z 143,A -152.6368,B 24.8861,C -1.4458,E1 24.7879,E2 599.0075} C_DIS
LIN {X -108.402,Y -68.4675,Z 143,A -150.3633,B 24.8856,C -1.4537,E1 24.7913,E2 596.7037} C_DIS
LIN {X -106.3986,Y -71.5421,Z 143,A -149.2854,B 24.8873,C -1.4228,E1 24.7928,E2 595.6941} C_DIS
LIN {X -104.6257,Y -74.1101,Z 143,A -147.6377,B 24.8869,C -1.4312,E1 24.7955,E2 594.0183} C_DIS
LIN {X -101.7664,Y -77.9898,Z 143,A -145.6801,B 24.8877,C -1.4165,E1 24.7987,E2 592.0862} C_DIS
LIN {X -99.6271,Y -80.705,Z 143,A -143.9208,B 24.8873,C -1.4229,E1 24.8019,E2 590.3034} C_DIS
LIN {X -96.9067,Y -83.9525,Z 143,A -141.9699,B 24.8874,C -1.4212,E1 24.8054,E2 588.3477} C_DIS
LIN {X -94.0155,Y -87.1776,Z 143,A -140.0125,B 24.8876,C -1.4178,E1 24.8091,E2 586.3896} C_DIS
LIN {X -90.9338,Y -90.3871,Z 143,A -138.052,B 24.8879,C -1.4121,E1 24.8129,E2 584.4342} C_DIS
LIN {X -87.9166,Y -93.3246,Z 143,A -136.1741,B 24.8881,C -1.4079,E1 24.8167,E2 582.5584} C_DIS
LIN {X -84.6382,Y -96.3084,Z 143,A -134.1548,B 24.8882,C -1.4058,E1 24.8209,E2 580.5363} C_DIS
LIN {X -81.1168,Y -99.2918,Z 143,A -132.3079,B 24.889,C -1.3914,E1 24.8248,E2 578.7165} C_DIS
LIN {X -78.5191,Y -101.3585,Z 143,A -130.6011,B 24.8886,C -1.3994,E1 24.8286,E2 576.9844} C_DIS
LIN {X -74.7217,Y -104.1897,Z 143,A -128.6775,B 24.8892,C -1.3864,E1 24.8329,E2 575.0851} C_DIS
LIN {X -72.008,Y -106.0833,Z 143,A -126.9957,B 24.8889,C -1.3937,E1 24.8368,E2 573.38} C_DIS
LIN {X -68.1552,Y -108.5991,Z 143,A -124.9462,B 24.889,C -1.3901,E1 24.8416,E2 571.3325} C_DIS
LIN {X -64.6126,Y -110.7436,Z 143,A -123.0378,B 24.889,C -1.3901,E1 24.8462,E2 569.4182} C_DIS
LIN {X -60.9042,Y -112.8252,Z 143,A -121.1478,B 24.8892,C -1.387,E1 24.8508,E2 567.5302} C_DIS
LIN {X -57.9915,Y -114.3474,Z 143,A -119.7933,B 24.8896,C -1.3796,E1 24.8542,E2 566.1897} C_DIS
LIN {X -55.0337,Y -115.8001,Z 143,A -118.2908,B 24.8896,C -1.3792,E1 24.8579,E2 564.6841} C_DIS
LIN {X -50.2193,Y -117.9697,Z 143,A -115.9897,B 24.8899,C -1.3737,E1 24.8638,E2 562.3908} C_DIS
LIN {X -46.1914,Y -119.6025,Z 143,A -114.0205,B 24.8899,C -1.3731,E1 24.8689,E2 560.4187} C_DIS
LIN {X -41.9333,Y -121.1608,Z 143,A -112.0485,B 24.8902,C -1.3686,E1 24.8741,E2 558.4534} C_DIS
LIN {X -38.9785,Y -122.1434,Z 143,A -110.5896,B 24.8901,C -1.3708,E1 24.878,E2 556.9867} C_DIS
LIN {X -35.6734,Y -123.1499,Z 143,A -108.8956,B 24.8897,C -1.3771,E1 24.8826,E2 555.2748} C_DIS
LIN {X -31.6368,Y -124.2477,Z 143,A -107.1745,B 24.8902,C -1.3686,E1 24.8872,E2 553.5714} C_DIS
LIN {X -28.4823,Y -125.0085,Z 143,A -105.7152,B 24.8902,C -1.3683,E1 24.8911,E2 552.1108} C_DIS
LIN {X -24.7039,Y -125.8114,Z 143,A -103.5811,B 24.8892,C -1.3879,E1 24.8971,E2 549.9276} C_DIS
LIN {X -21.1894,Y -126.4492,Z 143,A -102.0671,B 24.8894,C -1.3833,E1 24.9012,E2 548.4232} C_DIS
LIN {X -17.9522,Y -126.9494,Z 143,A -100.916,B 24.8902,C -1.3673,E1 24.9043,E2 547.3092} C_DIS
LIN {X -14.4868,Y -127.3932,Z 143,A -98.5992,B 24.8883,C -1.4051,E1 24.911,E2 544.901} C_DIS
LIN {X -9.1115,Y -127.8884,Z 143,A -96.424,B 24.8889,C -1.393,E1 24.917,E2 542.7536} C_DIS
LIN {X -4.8323,Y -128.1215,Z 143,A -95.3633,B 24.8911,C -1.3501,E1 24.9197,E2 541.7946} C_DIS
LIN {X -2.1559,Y -128.1944,Z 143,A -93.2451,B 24.8887,C -1.3969,E1 24.9259,E2 539.5652} C_DIS
LIN {X -2.1559,Y -128.1944,Z 143,A -93.2451,B 24.8887,C -1.3969,E1 24.9259,E2 539.5652} C_DIS
Enddeposition()
LIN {X 0.9052,Y -127.2215,Z 143,A -92.4367,B 24.1289,C -1.2281,E1 24.1602,E2 539.0586} C_DIS
Startdeposition()
$VEL.CP = VEL_PRINT
LIN {X -2.312,Y -127.2259,Z 143,A -95.1424,B 24.1317,C -1.1676,E1 24.1522,E2 541.9124} C_DIS
LIN {X -7.8373,Y -127.0051,Z 143,A -96.5742,B 24.1294,C -1.2175,E1 24.1486,E2 543.2224} C_DIS
LIN {X -13.1776,Y -126.5632,Z 143,A -99.1114,B 24.1297,C -1.2117,E1 24.1415,E2 545.7751} C_DIS
LIN {X -16.399,Y -126.1855,Z 143,A -101.2166,B 24.1311,C -1.1816,E1 24.1354,E2 547.9557} C_DIS
LIN {X -20.465,Y -125.5903,Z 143,A -102.4052,B 24.1296,C -1.2132,E1 24.1323,E2 549.0679} C_DIS
LIN {X -23.1905,Y -125.1175,Z 143,A -103.9722,B 24.1303,C -1.1985,E1 24.1279,E2 550.6727} C_DIS
LIN {X -27.2111,Y -124.3035,Z 143,A -105.7929,B 24.1302,C -1.2006,E1 24.1229,E2 552.4905} C_DIS
LIN {X -31.1861,Y -123.3657,Z 143,A -107.5262,B 24.1299,C -1.2065,E1 24.1183,E2 554.2117} C_DIS
LIN {X -34.4157,Y -122.504,Z 143,A -109.005,B 24.1298,C -1.2087,E1 24.1143,E2 555.6874} C_DIS
LIN {X -37.9083,Y -121.4705,Z 143,A -110.802,B 24.1301,C -1.2026,E1 24.1095,E2 557.5027} C_DIS
LIN {X -45.2567,Y -118.9281,Z 143,A -115.2254,B 24.1319,C -1.1634,E1 24.0976,E2 562.0314} C_DIS
LIN {X -51.5746,Y -116.3264,Z 143,A -117.0864,B 24.1291,C -1.2225,E1 24.0932,E2 563.7521} C_DIS
LIN {X -53.7533,Y -115.3357,Z 143,A -118.3098,B 24.1294,C -1.217,E1 24.09,E2 564.9921} C_DIS
LIN {X -56.5628,Y -113.9839,Z 143,A -119.766,B 24.1294,C -1.2163,E1 24.0863,E2 566.4538} C_DIS
LIN {X -61.1645,Y -111.5843,Z 143,A -122.095,B 24.1293,C -1.2198,E1 24.0806,E2 568.7811} C_DIS
LIN {X -64.7418,Y -109.5476,Z 143,A -124.4429,B 24.1302,C -1.1999,E1 24.0748,E2 571.1851} C_DIS
LIN {X -68.2629,Y -107.3891,Z 143,A -125.8089,B 24.129,C -1.2252,E1 24.0717,E2 572.4935} C_DIS
LIN {X -71.5575,Y -105.222,Z 143,A -127.7063,B 24.1291,C -1.2226,E1 24.0673,E2 574.4039} C_DIS
LIN {X -76.9212,Y -101.3672,Z 143,A -130.3766,B 24.1282,C -1.2416,E1 24.0614,E2 577.0372} C_DIS
LIN {X -82.0132,Y -97.2933,Z 143,A -133.6143,B 24.1286,C -1.2334,E1 24.0542,E2 580.3078} C_DIS
LIN {X -85.2213,Y -94.4963,Z 143,A -135.5776,B 24.1286,C -1.2351,E1 24.0501,E2 582.2749} C_DIS
LIN {X -88.3813,Y -91.5469,Z 143,A -137.5199,B 24.1283,C -1.2394,E1 24.0462,E2 584.2152} C_DIS
LIN {X -91.6356,Y -88.2897,Z 143,A -139.6148,B 24.1282,C -1.2429,E1 24.0421,E2 586.3106} C_DIS
LIN {X -94.5991,Y -85.1068,Z 143,A -141.5685,B 24.1279,C -1.2475,E1 24.0384,E2 588.262} C_DIS
LIN {X -97.4516,Y -81.8246,Z 143,A -143.5282,B 24.1277,C -1.252,E1 24.0349,E2 590.2198} C_DIS
LIN {X -100.3146,Y -78.2893,Z 143,A -146.1364,B 24.1287,C -1.2321,E1 24.0303,E2 592.8897} C_DIS
LIN {X -103.2256,Y -74.4087,Z 143,A -148.7946,B 24.1294,C -1.2169,E1 24.0259,E2 595.5988} C_DIS
LIN {X -107.2234,Y -68.5217,Z 143,A -150.9511,B 24.1268,C -1.2713,E1 24.0228,E2 597.6329} C_DIS
LIN {X -109.4883,Y -64.8422,Z 143,A -152.9911,B 24.1268,C -1.2723,E1 24.0198,E2 599.6813} C_DIS
LIN {X -111.6592,Y -61.0271,Z 143,A -154.7518,B 24.126,C -1.2873,E1 24.0174,E2 601.4148} C_DIS
LIN {X -112.8543,Y -58.785,Z 143,A -155.9812,B 24.126,C -1.2867,E1 24.0158,E2 602.6524} C_DIS
LIN {X -115.4645,Y -53.4748,Z 143,A -158.3766,B 24.125,C -1.3062,E1 24.0129,E2 605.0134} C_DIS
LIN {X -116.768,Y -50.5652,Z 143,A -160.1167,B 24.1255,C -1.2969,E1 24.0109,E2 606.7864} C_DIS
LIN {X -118.0169,Y -47.5775,Z 143,A -161.5862,B 24.1253,C -1.3006,E1 24.0093,E2 608.2551} C_DIS
LIN {X -119.1786,Y -44.588,Z 143,A -163.0556,B 24.1251,C -1.3038,E1 24.0079,E2 609.7253} C_DIS
LIN {X -120.307,Y -41.4476,Z 143,A -164.5823,B 24.125,C -1.3073,E1 24.0065,E2 611.2525} C_DIS
LIN {X -121.6162,Y -37.4323,Z 143,A -167.1138,B 24.1261,C -1.2856,E1 24.0043,E2 613.8524} C_DIS
LIN {X -122.9379,Y -32.8318,Z 143,A -168.6718,B 24.1244,C -1.3182,E1 24.0032,E2 615.3395} C_DIS
LIN {X -123.8387,Y -29.2569,Z 143,A -171.0107,B 24.1256,C -1.2939,E1 24.0017,E2 617.7526} C_DIS
LIN {X -124.8998,Y -24.3292,Z 143,A -172.4461,B 24.1234,C -1.3373,E1 24.0009,E2 619.0899} C_DIS
LIN {X -125.5674,Y -20.6063,Z 143,A -174.4429,B 24.1238,C -1.3299,E1 23.9999,E2 621.1174} C_DIS
LIN {X -126.1645,Y -16.5593,Z 143,A -176.1689,B 24.1232,C -1.3408,E1 23.9993,E2 622.8271} C_DIS
LIN {X -126.5795,Y -13.0259,Z 143,A -177.9175,B 24.1232,C -1.3396,E1 23.9987,E2 624.5897} C_DIS
LIN {X -126.9469,Y -8.7452,Z 143,A -179.7563,B 24.1227,C -1.35,E1 23.9983,E2 626.4143} C_DIS
LIN {X -127.1489,Y -4.989,Z 143,A 178.5554,B 24.1224,C -1.3557,E1 23.9981,E2 628.099} C_DIS
LIN {X -127.2455,Y -0.836,Z 143,A 176.785,B 24.1219,C -1.3662,E1 23.9981,E2 629.8548} C_DIS
LIN {X -127.2213,Y 2.5899,Z 143,A 174.9927,B 24.1222,C -1.3603,E1 23.9981,E2 631.6728} C_DIS
LIN {X -127.0753,Y 6.6063,Z 143,A 173.244,B 24.1217,C -1.3689,E1 23.9983,E2 633.4114} C_DIS
LIN {X -126.7972,Y 10.6858,Z 143,A 171.4285,B 24.1214,C -1.376,E1 23.9987,E2 635.2206} C_DIS
LIN {X -126.392,Y 14.7266,Z 143,A 169.361,B 24.1216,C -1.3716,E1 23.9993,E2 637.3118} C_DIS
LIN {X -125.8831,Y 18.587,Z 143,A 167.7443,B 24.121,C -1.3832,E1 23.9999,E2 638.91} C_DIS
LIN {X -125.27,Y 22.3409,Z 143,A 166.0837,B 24.1206,C -1.3911,E1 24.0007,E2 640.5616} C_DIS
Enddeposition()
END
